C05451=1075.122,-81.429,-56.571,173.054,21.010,153.734
C05452=1075.129,-81.150,-56.583,173.055,21.011,153.734
C05453=1075.136,-80.901,-56.593,173.057,21.013,153.734
C05454=1075.142,-80.652,-56.604,173.058,21.015,153.734
C05455=1075.148,-80.401,-56.615,173.060,21.016,153.734
C05456=1075.154,-80.152,-56.626,173.061,21.018,153.734
C05457=1075.160,-79.903,-56.637,173.063,21.019,153.734
C05458=1075.166,-79.652,-56.647,173.064,21.020,153.734
C05459=1075.172,-79.403,-56.658,173.066,21.023,153.734
C05460=1075.178,-79.153,-56.669,173.068,21.024,153.734
C05461=1075.184,-78.903,-56.680,173.069,21.026,153.734
C05462=1075.190,-78.654,-56.690,173.071,21.028,153.734
C05463=1075.196,-78.404,-56.701,173.072,21.029,153.734
C05464=1075.203,-78.154,-56.712,173.074,21.030,153.734
C05465=1075.208,-77.904,-56.723,173.075,21.032,153.734
C05466=1075.214,-77.655,-56.734,173.077,21.034,153.734
C05467=1075.220,-77.405,-56.745,173.078,21.035,153.734
C05468=1075.226,-77.155,-56.756,173.080,21.037,153.735
C05469=1075.232,-76.906,-56.767,173.081,21.039,153.735
C05470=1075.239,-76.656,-56.778,173.083,21.040,153.735
C05471=1075.245,-76.406,-56.789,173.084,21.042,153.735
C05472=1075.250,-76.157,-56.800,173.086,21.044,153.735
C05473=1075.257,-75.907,-56.811,173.087,21.045,153.735
C05474=1075.263,-75.658,-56.822,173.088,21.047,153.735
C05475=1075.269,-75.408,-56.833,173.090,21.048,153.735
C05476=1075.275,-75.158,-56.845,173.092,21.050,153.735
C05477=1075.281,-74.909,-56.855,173.093,21.052,153.735
C05478=1075.287,-74.659,-56.867,173.094,21.053,153.735
C05479=1075.293,-74.409,-56.878,173.096,21.055,153.735
C05480=1075.298,-74.160,-56.888,173.097,21.057,153.735
C05481=1075.305,-73.909,-56.900,173.099,21.058,153.735
C05482=1075.310,-73.660,-56.911,173.100,21.060,153.736
C05483=1075.316,-73.410,-56.921,173.102,21.061,153.736
C05484=1075.323,-73.160,-56.933,173.103,21.063,153.736
C05485=1075.329,-72.911,-56.944,173.105,21.065,153.736
C05486=1075.334,-72.662,-56.955,173.106,21.067,153.736
C05487=1075.341,-72.412,-56.966,173.107,21.068,153.736
C05488=1075.346,-72.162,-56.977,173.109,21.070,153.736
C05489=1075.352,-71.913,-56.988,173.110,21.072,153.736
C05490=1075.358,-71.662,-57.000,173.113,21.074,153.736
C05491=1075.364,-71.413,-57.012,173.114,21.075,153.736
C05492=1075.370,-71.163,-57.023,173.115,21.077,153.736
C05493=1075.376,-70.914,-57.034,173.117,21.079,153.737
C05494=1075.382,-70.664,-57.045,173.118,21.081,153.737
C05495=1075.388,-70.414,-57.056,173.120,21.083,153.737
C05496=1075.394,-70.165,-57.067,173.121,21.084,153.737
C05497=1075.399,-69.915,-57.079,173.123,21.086,153.737
C05498=1075.405,-69.665,-57.090,173.124,21.088,153.737
C05499=1075.411,-69.416,-57.101,173.125,21.089,153.737
C05500=1075.417,-69.165,-57.112,173.127,21.091,153.737
C05501=1075.424,-68.917,-57.124,173.128,21.093,153.737
C05502=1075.429,-68.667,-57.135,173.130,21.095,153.737
C05503=1075.436,-68.417,-57.146,173.131,21.096,153.738
C05504=1075.441,-68.167,-57.157,173.132,21.098,153.738
C05505=1075.447,-67.917,-57.169,173.134,21.100,153.738
C05506=1075.453,-67.668,-57.180,173.135,21.102,153.738
C05507=1075.459,-67.418,-57.192,173.137,21.103,153.738
C05508=1075.465,-67.169,-57.203,173.138,21.105,153.738
C05509=1075.470,-66.919,-57.215,173.140,21.107,153.738
C05510=1075.477,-66.669,-57.226,173.142,21.109,153.738
C05511=1075.482,-66.419,-57.237,173.143,21.111,153.738
C05512=1075.489,-66.170,-57.249,173.145,21.112,153.738
C05513=1075.495,-65.893,-57.261,173.146,21.114,153.738
C05514=1075.502,-65.617,-57.274,173.148,21.116,153.739
C05515=1075.509,-65.341,-57.287,173.149,21.118,153.739
C05516=1075.515,-65.064,-57.299,173.151,21.121,153.739
C05517=1075.521,-64.814,-57.310,173.153,21.122,153.739
C05518=1075.527,-64.565,-57.322,173.154,21.124,153.739
C05519=1075.534,-64.315,-57.333,173.155,21.126,153.739
C05520=1075.539,-64.066,-57.345,173.157,21.127,153.739
C05521=1075.545,-63.815,-57.356,173.158,21.129,153.739
C05522=1075.551,-63.566,-57.367,173.160,21.131,153.739
C05523=1075.558,-63.316,-57.379,173.161,21.133,153.740
C05524=1075.563,-63.067,-57.390,173.162,21.135,153.740
C05525=1075.569,-62.817,-57.403,173.164,21.136,153.740
C05526=1075.575,-62.567,-57.414,173.165,21.138,153.740
C05527=1075.581,-62.317,-57.425,173.167,21.140,153.740
C05528=1075.587,-62.068,-57.436,173.169,21.142,153.740
C05529=1075.593,-61.818,-57.448,173.170,21.144,153.740
C05530=1075.599,-61.569,-57.460,173.172,21.146,153.740
C05531=1075.605,-61.319,-57.471,173.173,21.147,153.740
C05532=1075.612,-61.069,-57.483,173.175,21.149,153.741
C05533=1075.617,-60.819,-57.495,173.176,21.151,153.741
C05534=1075.624,-60.570,-57.506,173.177,21.153,153.741
C05535=1075.629,-60.320,-57.517,173.179,21.154,153.741
C05536=1075.636,-60.071,-57.529,173.180,21.156,153.741
C05537=1075.641,-59.821,-57.541,173.181,21.158,153.741
C05538=1075.648,-59.571,-57.553,173.183,21.160,153.741
C05539=1075.654,-59.321,-57.564,173.184,21.162,153.741
C05540=1075.660,-59.072,-57.576,173.186,21.164,153.742
C05541=1075.666,-58.822,-57.587,173.187,21.165,153.742
C05542=1075.672,-58.573,-57.599,173.189,21.168,153.742
C05543=1075.678,-58.323,-57.610,173.191,21.170,153.742
C05544=1075.683,-58.074,-57.622,173.192,21.172,153.742
C05545=1075.690,-57.823,-57.634,173.194,21.173,153.742
C05546=1075.696,-57.574,-57.646,173.195,21.175,153.742
C05547=1075.702,-57.325,-57.657,173.196,21.177,153.742
C05548=1075.708,-57.074,-57.669,173.198,21.178,153.742
C05549=1075.715,-56.825,-57.681,173.199,21.180,153.743
C05550=1075.720,-56.575,-57.692,173.201,21.182,153.743
C05551=1075.726,-56.326,-57.704,173.202,21.184,153.743
C05552=1075.732,-56.077,-57.716,173.203,21.186,153.743
C05553=1075.739,-55.826,-57.727,173.205,21.188,153.743
C05554=1075.745,-55.577,-57.739,173.206,21.190,153.743
C05555=1075.750,-55.327,-57.751,173.208,21.192,153.743
C05556=1075.757,-55.078,-57.763,173.210,21.193,153.743
C05557=1075.764,-54.828,-57.775,173.211,21.195,153.743
C05558=1075.769,-54.578,-57.786,173.213,21.197,153.744
C05559=1075.775,-54.329,-57.798,173.214,21.199,153.744
C05560=1075.782,-54.079,-57.810,173.215,21.201,153.744
C05561=1075.787,-53.829,-57.822,173.217,21.203,153.744
C05562=1075.794,-53.580,-57.833,173.218,21.205,153.744
C05563=1075.800,-53.330,-57.845,173.219,21.207,153.744
C05564=1075.806,-53.081,-57.858,173.221,21.208,153.744
C05565=1075.812,-52.831,-57.869,173.222,21.210,153.744
C05566=1075.819,-52.581,-57.881,173.225,21.212,153.745
C05567=1075.824,-52.332,-57.893,173.226,21.214,153.745
C05568=1075.830,-52.082,-57.904,173.227,21.216,153.745
C05569=1075.837,-51.832,-57.916,173.229,21.218,153.745
C05570=1075.843,-51.582,-57.929,173.230,21.220,153.745
C05571=1075.849,-51.333,-57.940,173.232,21.222,153.745
C05572=1075.854,-51.083,-57.952,173.233,21.224,153.745
C05573=1075.861,-50.833,-57.964,173.234,21.225,153.746
C05574=1075.867,-50.584,-57.976,173.236,21.227,153.746
C05575=1075.873,-50.335,-57.988,173.237,21.229,153.746
C05576=1075.879,-50.084,-58.000,173.238,21.231,153.746
C05577=1075.886,-49.810,-58.013,173.241,21.233,153.746
C05578=1075.892,-49.534,-58.026,173.242,21.236,153.746
C05579=1075.899,-49.259,-58.040,173.243,21.238,153.746
C05580=1075.905,-48.984,-58.053,173.245,21.240,153.747
C05581=1075.912,-48.699,-58.067,173.247,21.242,153.747
C05582=1075.919,-48.414,-58.080,173.248,21.245,153.747
C05583=1075.926,-48.130,-58.095,173.250,21.247,153.747
C05584=1075.932,-47.846,-58.108,173.251,21.249,153.747
C05585=1075.938,-47.596,-58.120,173.253,21.251,153.747
C05586=1075.944,-47.346,-58.133,173.254,21.253,153.748
C05587=1075.950,-47.097,-58.145,173.256,21.255,153.748
C05588=1075.956,-46.847,-58.157,173.258,21.257,153.748
C05589=1075.962,-46.597,-58.169,173.259,21.259,153.748
C05590=1075.968,-46.348,-58.181,173.260,21.261,153.748
C05591=1075.974,-46.098,-58.193,173.262,21.263,153.748
C05592=1075.980,-45.848,-58.206,173.263,21.265,153.748
C05593=1075.986,-45.599,-58.217,173.264,21.267,153.749
C05594=1075.992,-45.349,-58.230,173.266,21.269,153.749
C05595=1075.998,-45.099,-58.242,173.267,21.271,153.749
C05596=1076.004,-44.850,-58.254,173.269,21.273,153.749
C05597=1076.010,-44.601,-58.266,173.271,21.275,153.749
C05598=1076.015,-44.351,-58.279,173.272,21.277,153.749
C05599=1076.022,-44.101,-58.291,173.273,21.279,153.750
C05600=1076.028,-43.851,-58.304,173.275,21.281,153.750
C05601=1076.033,-43.602,-58.316,173.276,21.283,153.750
C05602=1076.040,-43.352,-58.328,173.277,21.285,153.750
C05603=1076.046,-43.103,-58.340,173.279,21.287,153.750
C05604=1076.052,-42.853,-58.353,173.280,21.289,153.750
C05605=1076.058,-42.604,-58.364,173.282,21.291,153.750
C05606=1076.064,-42.354,-58.377,173.284,21.293,153.751
C05607=1076.070,-42.104,-58.389,173.285,21.295,153.751
C05608=1076.076,-41.854,-58.401,173.286,21.297,153.751
C05609=1076.082,-41.605,-58.414,173.288,21.299,153.751
C05610=1076.087,-41.355,-58.426,173.289,21.302,153.751
C05611=1076.094,-41.106,-58.438,173.290,21.304,153.752
C05612=1076.100,-40.856,-58.451,173.291,21.306,153.752
C05613=1076.106,-40.606,-58.463,173.293,21.308,153.752
C05614=1076.112,-40.356,-58.476,173.295,21.310,153.752
C05615=1076.118,-40.107,-58.487,173.296,21.312,153.752
C05616=1076.124,-39.857,-58.500,173.298,21.314,153.752
C05617=1076.130,-39.608,-58.513,173.299,21.316,153.752
C05618=1076.136,-39.358,-58.525,173.300,21.318,153.753
C05619=1076.142,-39.108,-58.537,173.302,21.320,153.753
C05620=1076.148,-38.858,-58.550,173.303,21.322,153.753
C05621=1076.154,-38.610,-58.562,173.304,21.324,153.753
C05622=1076.160,-38.360,-58.575,173.307,21.326,153.753
C05623=1076.166,-38.110,-58.587,173.308,21.329,153.754
C05624=1076.172,-37.860,-58.600,173.309,21.330,153.754
C05625=1076.178,-37.610,-58.612,173.310,21.332,153.754
C05626=1076.183,-37.361,-58.624,173.312,21.334,153.754
C05627=1076.189,-37.111,-58.637,173.313,21.336,153.754
C05628=1076.196,-36.862,-58.650,173.315,21.338,153.754
C05629=1076.202,-36.612,-58.663,173.316,21.341,153.755
C05630=1076.207,-36.362,-58.675,173.318,21.343,153.755
C05631=1076.213,-36.113,-58.687,173.319,21.345,153.755
C05632=1076.219,-35.863,-58.700,173.321,21.347,153.755
C05633=1076.225,-35.613,-58.713,173.322,21.349,153.755
C05634=1076.231,-35.364,-58.726,173.323,21.352,153.755
C05635=1076.237,-35.115,-58.738,173.324,21.353,153.756
C05636=1076.243,-34.865,-58.750,173.326,21.355,153.756
C05637=1076.248,-34.620,-58.763,173.327,21.357,153.756
C05638=1076.254,-34.375,-58.775,173.328,21.359,153.756
C05639=1076.260,-34.131,-58.787,173.330,21.362,153.756
C05640=1076.265,-33.886,-58.800,173.332,21.364,153.757
C05641=1076.272,-33.641,-58.813,173.333,21.366,153.757
C05642=1076.278,-33.397,-58.825,173.335,21.368,153.757
C05643=1076.283,-33.152,-58.837,173.336,21.370,153.757
C05644=1076.289,-32.907,-58.850,173.337,21.372,153.757
C05645=1076.295,-32.658,-58.862,173.338,21.375,153.757
C05646=1076.301,-32.408,-58.875,173.340,21.376,153.758
C05647=1076.307,-32.158,-58.888,173.341,21.378,153.758
C05648=1076.313,-31.909,-58.900,173.342,21.380,153.758
C05649=1076.319,-31.659,-58.913,173.345,21.383,153.758
C05650=1076.325,-31.409,-58.926,173.346,21.385,153.758
C05651=1076.331,-31.159,-58.939,173.347,21.387,153.759
C05652=1076.337,-30.910,-58.951,173.348,21.389,153.759
C05653=1076.343,-30.661,-58.964,173.350,21.391,153.759
C05654=1076.349,-30.411,-58.977,173.351,21.394,153.759
C05655=1076.355,-30.162,-58.990,173.352,21.396,153.759
C05656=1076.361,-29.912,-59.003,173.355,21.398,153.759
C05657=1076.367,-29.662,-59.015,173.356,21.400,153.760
C05658=1076.373,-29.413,-59.028,173.357,21.402,153.760
C05659=1076.379,-29.163,-59.041,173.358,21.404,153.760
C05660=1076.385,-28.913,-59.054,173.360,21.406,153.760
C05661=1076.391,-28.664,-59.067,173.361,21.408,153.760
C05662=1076.397,-28.414,-59.079,173.362,21.411,153.761
C05663=1076.403,-28.165,-59.093,173.364,21.413,153.761
C05664=1076.409,-27.915,-59.105,173.366,21.415,153.761
C05665=1076.415,-27.666,-59.119,173.367,21.417,153.761
C05666=1076.421,-27.416,-59.131,173.368,21.420,153.761
C05667=1076.427,-27.166,-59.144,173.370,21.421,153.762
C05668=1076.433,-26.917,-59.157,173.371,21.423,153.762
C05669=1076.439,-26.667,-59.169,173.372,21.425,153.762
C05670=1076.445,-26.417,-59.183,173.374,21.428,153.762
C05671=1076.451,-26.167,-59.195,173.376,21.430,153.762
C05672=1076.456,-25.919,-59.209,173.377,21.433,153.763
C05673=1076.462,-25.669,-59.221,173.378,21.435,153.763
C05674=1076.468,-25.419,-59.235,173.380,21.437,153.763
C05675=1076.474,-25.170,-59.247,173.381,21.439,153.763
C05676=1076.480,-24.920,-59.260,173.382,21.441,153.763
C05677=1076.486,-24.670,-59.274,173.384,21.443,153.763
C05678=1076.492,-24.421,-59.287,173.385,21.446,153.764
C05679=1076.498,-24.171,-59.299,173.387,21.448,153.764
C05680=1076.504,-23.922,-59.313,173.388,21.450,153.764
C05681=1076.509,-23.672,-59.327,173.389,21.452,153.764
C05682=1076.515,-23.422,-59.339,173.391,21.454,153.764
C05683=1076.521,-23.173,-59.352,173.392,21.457,153.765
C05684=1076.527,-22.923,-59.365,173.394,21.459,153.765
C05685=1076.534,-22.674,-59.378,173.395,21.461,153.765
C05686=1076.539,-22.424,-59.391,173.397,21.464,153.765
C05687=1076.545,-22.174,-59.405,173.398,21.466,153.766
C05688=1076.551,-21.925,-59.418,173.399,21.468,153.766
C05689=1076.557,-21.675,-59.430,173.400,21.470,153.766
C05690=1076.563,-21.426,-59.444,173.402,21.472,153.766
C05691=1076.569,-21.176,-59.457,173.404,21.475,153.766
C05692=1076.575,-20.927,-59.470,173.405,21.477,153.767
C05693=1076.581,-20.677,-59.483,173.407,21.479,153.767
C05694=1076.586,-20.427,-59.497,173.408,21.481,153.767
C05695=1076.592,-20.178,-59.510,173.409,21.483,153.767
C05696=1076.599,-19.929,-59.523,173.410,21.486,153.767
C05697=1076.604,-19.679,-59.536,173.412,21.488,153.768
C05698=1076.610,-19.429,-59.549,173.414,21.490,153.768
C05699=1076.616,-19.180,-59.563,173.415,21.493,153.768
C05700=1076.622,-18.930,-59.575,173.416,21.494,153.768
C05701=1076.628,-18.680,-59.590,173.417,21.497,153.768
C05702=1076.634,-18.430,-59.603,173.419,21.499,153.769
C05703=1076.641,-18.181,-59.616,173.420,21.501,153.769
C05704=1076.646,-17.931,-59.629,173.422,21.504,153.769
C05705=1076.653,-17.656,-59.643,173.424,21.506,153.769
C05706=1076.659,-17.380,-59.658,173.425,21.508,153.770
C05707=1076.666,-17.105,-59.673,173.427,21.511,153.770
C05708=1076.673,-16.829,-59.688,173.428,21.513,153.770
C05709=1076.679,-16.579,-59.701,173.429,21.516,153.770
C05710=1076.684,-16.330,-59.714,173.431,21.517,153.770
C05711=1076.690,-16.080,-59.728,173.433,21.520,153.771
C05712=1076.696,-15.831,-59.741,173.434,21.522,153.771
C05713=1076.702,-15.581,-59.755,173.435,21.524,153.771
C05714=1076.708,-15.331,-59.768,173.436,21.527,153.771
C05715=1076.715,-15.082,-59.781,173.438,21.529,153.771
C05716=1076.720,-14.832,-59.795,173.439,21.531,153.772
C05717=1076.726,-14.583,-59.808,173.441,21.534,153.772
C05718=1076.732,-14.333,-59.822,173.442,21.536,153.772
C05719=1076.738,-14.083,-59.835,173.444,21.538,153.772
C05720=1076.743,-13.834,-59.849,173.445,21.541,153.773
C05721=1076.749,-13.584,-59.862,173.446,21.542,153.773
C05722=1076.755,-13.335,-59.876,173.447,21.545,153.773
C05723=1076.761,-13.086,-59.889,173.449,21.547,153.773
C05724=1076.767,-12.836,-59.903,173.451,21.550,153.773
C05725=1076.773,-12.586,-59.916,173.452,21.552,153.774
C05726=1076.779,-12.336,-59.930,173.453,21.554,153.774
C05727=1076.785,-12.087,-59.943,173.455,21.556,153.774
C05728=1076.790,-11.837,-59.957,173.456,21.559,153.774
C05729=1076.797,-11.588,-59.970,173.457,21.561,153.775
C05730=1076.802,-11.338,-59.984,173.459,21.564,153.775
C05731=1076.808,-11.089,-59.997,173.460,21.566,153.775
C05732=1076.814,-10.839,-60.011,173.462,21.568,153.775
C05733=1076.820,-10.589,-60.025,173.463,21.570,153.776
C05734=1076.826,-10.340,-60.038,173.464,21.572,153.776
C05735=1076.832,-10.091,-60.052,173.465,21.575,153.776
C05736=1076.838,-9.841,-60.066,173.468,21.577,153.776
C05737=1076.844,-9.592,-60.079,173.469,21.580,153.776
C05738=1076.849,-9.342,-60.093,173.470,21.582,153.777
C05739=1076.856,-9.093,-60.106,173.471,21.584,153.777
C05740=1076.862,-8.843,-60.120,173.473,21.586,153.777
C05741=1076.867,-8.593,-60.134,173.474,21.589,153.777
C05742=1076.873,-8.344,-60.147,173.476,21.591,153.777
C05743=1076.879,-8.094,-60.161,173.477,21.593,153.778
C05744=1076.885,-7.845,-60.174,173.479,21.595,153.778
C05745=1076.891,-7.595,-60.189,173.480,21.598,153.778
C05746=1076.897,-7.345,-60.202,173.481,21.600,153.778
C05747=1076.903,-7.096,-60.216,173.483,21.603,153.779
C05748=1076.909,-6.847,-60.229,173.485,21.605,153.779
C05749=1076.914,-6.597,-60.243,173.486,21.607,153.779
C05750=1076.921,-6.347,-60.257,173.487,21.609,153.779
C05751=1076.927,-6.097,-60.270,173.488,21.612,153.779
C05752=1076.932,-5.848,-60.284,173.489,21.614,153.780
C05753=1076.938,-5.599,-60.298,173.492,21.616,153.780
C05754=1076.945,-5.348,-60.312,173.493,21.619,153.780
C05755=1076.950,-5.099,-60.326,173.494,21.621,153.780
C05756=1076.957,-4.850,-60.340,173.495,21.623,153.781
C05757=1076.962,-4.601,-60.354,173.497,21.625,153.781
C05758=1076.969,-4.351,-60.367,173.498,21.628,153.781
C05759=1076.974,-4.101,-60.381,173.500,21.630,153.781
C05760=1076.980,-3.851,-60.395,173.501,21.633,153.782
C05761=1076.986,-3.602,-60.408,173.503,21.634,153.782
C05762=1076.992,-3.353,-60.423,173.504,21.637,153.782
C05763=1076.998,-3.103,-60.437,173.505,21.639,153.782
C05764=1077.004,-2.854,-60.450,173.506,21.641,153.782
C05765=1077.010,-2.604,-60.464,173.508,21.644,153.783
C05766=1077.016,-2.354,-60.478,173.510,21.646,153.783
C05767=1077.021,-2.104,-60.492,173.511,21.649,153.783
C05768=1077.027,-1.855,-60.507,173.512,21.651,153.783
C05769=1077.033,-1.578,-60.522,173.514,21.654,153.784
C05770=1077.040,-1.300,-60.538,173.515,21.657,153.784
C05771=1077.046,-1.023,-60.553,173.516,21.659,153.784
C05772=1077.053,-0.746,-60.569,173.518,21.662,153.785
C05773=1077.058,-0.496,-60.583,173.520,21.664,153.785
C05774=1077.064,-0.247,-60.597,173.521,21.666,153.785
C05775=1077.070,0.002,-60.610,173.522,21.669,153.785
C05776=1077.076,0.252,-60.625,173.524,21.671,153.785
C05777=1077.082,0.501,-60.639,173.526,21.674,153.786
C05778=1077.088,0.751,-60.653,173.527,21.676,153.786
C05779=1077.093,1.000,-60.667,173.528,21.678,153.786
C05780=1077.099,1.251,-60.681,173.529,21.681,153.786
C05781=1077.105,1.500,-60.696,173.531,21.683,153.787
C05782=1077.110,1.749,-60.710,173.533,21.685,153.787
C05783=1077.117,1.999,-60.723,173.534,21.688,153.787
C05784=1077.123,2.248,-60.738,173.535,21.690,153.787
C05785=1077.128,2.498,-60.752,173.536,21.692,153.788
C05786=1077.134,2.747,-60.766,173.537,21.695,153.788
C05787=1077.140,2.997,-60.781,173.540,21.698,153.788
C05788=1077.146,3.247,-60.794,173.541,21.700,153.788
C05789=1077.151,3.496,-60.808,173.542,21.702,153.789
C05790=1077.158,3.746,-60.823,173.543,21.705,153.789
C05791=1077.163,3.995,-60.837,173.545,21.707,153.789
C05792=1077.170,4.244,-60.851,173.547,21.709,153.789
C05793=1077.176,4.494,-60.865,173.548,21.711,153.789
C05794=1077.181,4.744,-60.879,173.549,21.714,153.790
C05795=1077.187,4.993,-60.894,173.550,21.716,153.790
C05796=1077.193,5.243,-60.908,173.552,21.718,153.790
C05797=1077.199,5.492,-60.923,173.554,21.721,153.790
C05798=1077.204,5.742,-60.936,173.555,21.724,153.791
C05799=1077.211,5.991,-60.951,173.556,21.726,153.791
C05800=1077.216,6.241,-60.965,173.557,21.728,153.791
C05801=1077.222,6.490,-60.979,173.559,21.730,153.792
C05802=1077.228,6.740,-60.994,173.560,21.732,153.792
C05803=1077.234,6.990,-61.008,173.562,21.735,153.792
C05804=1077.239,7.239,-61.022,173.563,21.738,153.792
C05805=1077.245,7.489,-61.037,173.565,21.740,153.792
C05806=1077.252,7.738,-61.051,173.566,21.742,153.793
C05807=1077.258,7.988,-61.065,173.567,21.745,153.793
C05808=1077.264,8.237,-61.079,173.569,21.747,153.793
C05809=1077.269,8.486,-61.093,173.570,21.750,153.793
C05810=1077.276,8.736,-61.108,173.572,21.752,153.794
C05811=1077.281,8.985,-61.123,173.573,21.754,153.794
C05812=1077.288,9.235,-61.137,173.574,21.756,153.794
C05813=1077.293,9.484,-61.152,173.576,21.759,153.794
C05814=1077.299,9.735,-61.166,173.577,21.761,153.795
C05815=1077.305,9.983,-61.181,173.579,21.764,153.795
C05816=1077.311,10.233,-61.194,173.580,21.766,153.795
C05817=1077.317,10.483,-61.209,173.581,21.768,153.795
C05818=1077.323,10.732,-61.224,173.583,21.771,153.796
C05819=1077.329,10.982,-61.238,173.585,21.773,153.796
C05820=1077.335,11.231,-61.253,173.586,21.775,153.796
C05821=1077.341,11.481,-61.267,173.587,21.778,153.796
C05822=1077.347,11.730,-61.282,173.588,21.780,153.797
C05823=1077.353,11.980,-61.296,173.590,21.783,153.797
C05824=1077.358,12.229,-61.310,173.592,21.785,153.797
C05825=1077.365,12.479,-61.325,173.593,21.787,153.797
C05826=1077.371,12.728,-61.340,173.594,21.790,153.798
C05827=1077.376,12.978,-61.354,173.595,21.792,153.798
C05828=1077.382,13.227,-61.369,173.598,21.794,153.798
C05829=1077.388,13.476,-61.383,173.599,21.797,153.798
C05830=1077.394,13.726,-61.397,173.600,21.799,153.799
C05831=1077.400,13.975,-61.412,173.601,21.801,153.799
C05832=1077.406,14.225,-61.427,173.602,21.804,153.799
C05833=1077.413,14.505,-61.443,173.604,21.807,153.799
C05834=1077.419,14.783,-61.460,173.606,21.809,153.800
C05835=1077.426,15.063,-61.476,173.608,21.812,153.800
C05836=1077.432,15.342,-61.493,173.609,21.814,153.800
C05837=1077.438,15.592,-61.507,173.610,21.817,153.800
C05838=1077.444,15.842,-61.522,173.612,21.819,153.801
C05839=1077.450,16.091,-61.536,173.614,21.822,153.801
C05840=1077.456,16.340,-61.551,173.615,21.824,153.801
C05841=1077.461,16.590,-61.566,173.616,21.827,153.801
C05842=1077.467,16.840,-61.581,173.617,21.829,153.802
C05843=1077.473,17.089,-61.595,173.619,21.832,153.802
C05844=1077.480,17.338,-61.610,173.620,21.834,153.802
C05845=1077.485,17.587,-61.625,173.622,21.836,153.802
C05846=1077.491,17.838,-61.640,173.623,21.838,153.803
C05847=1077.496,18.087,-61.654,173.625,21.841,153.803
C05848=1077.503,18.337,-61.669,173.626,21.844,153.803
C05849=1077.509,18.586,-61.684,173.628,21.846,153.803
C05850=1077.514,18.836,-61.699,173.629,21.848,153.804
C05851=1077.520,19.084,-61.714,173.630,21.851,153.804
C05852=1077.526,19.335,-61.728,173.632,21.853,153.804
C05853=1077.532,19.584,-61.743,173.633,21.855,153.804
C05854=1077.538,19.834,-61.758,173.635,21.858,153.805
C05855=1077.543,20.083,-61.773,173.636,21.860,153.805
C05856=1077.550,20.332,-61.788,173.637,21.862,153.805
C05857=1077.555,20.581,-61.802,173.639,21.865,153.805
C05858=1077.561,20.831,-61.818,173.640,21.868,153.806
C05859=1077.567,21.080,-61.832,173.642,21.870,153.806
C05860=1077.573,21.330,-61.848,173.643,21.872,153.806
C05861=1077.578,21.579,-61.863,173.644,21.874,153.806
C05862=1077.584,21.829,-61.877,173.646,21.877,153.807
C05863=1077.590,22.079,-61.892,173.647,21.880,153.807
C05864=1077.596,22.328,-61.907,173.649,21.882,153.807
C05865=1077.602,22.578,-61.922,173.650,21.884,153.807
C05866=1077.607,22.827,-61.937,173.652,21.887,153.808
C05867=1077.614,23.077,-61.952,173.653,21.890,153.808
C05868=1077.619,23.326,-61.967,173.655,21.892,153.808
C05869=1077.625,23.576,-61.982,173.656,21.894,153.808
C05870=1077.631,23.825,-61.997,173.657,21.896,153.809
C05871=1077.637,24.075,-62.012,173.659,21.899,153.809
C05872=1077.643,24.324,-62.027,173.660,21.901,153.809
C05873=1077.649,24.573,-62.042,173.662,21.904,153.809
C05874=1077.654,24.823,-62.057,173.663,21.906,153.810
C05875=1077.660,25.072,-62.072,173.665,21.909,153.810
C05876=1077.666,25.322,-62.087,173.666,21.911,153.810
C05877=1077.672,25.572,-62.102,173.667,21.913,153.810
C05878=1077.678,25.821,-62.117,173.669,21.916,153.811
C05879=1077.684,26.070,-62.133,173.670,21.918,153.811
C05880=1077.690,26.320,-62.148,173.672,21.921,153.811
C05881=1077.695,26.569,-62.163,173.673,21.923,153.811
C05882=1077.702,26.819,-62.178,173.674,21.926,153.812
C05883=1077.707,27.068,-62.193,173.676,21.928,153.812
C05884=1077.713,27.318,-62.208,173.678,21.930,153.812
C05885=1077.719,27.567,-62.223,173.679,21.933,153.812
C05886=1077.725,27.817,-62.239,173.680,21.935,153.813
C05887=1077.731,28.066,-62.253,173.682,21.937,153.813
C05888=1077.737,28.316,-62.269,173.683,21.940,153.813
C05889=1077.743,28.565,-62.284,173.685,21.943,153.813
C05890=1077.748,28.815,-62.300,173.686,21.945,153.814
C05891=1077.755,29.064,-62.315,173.687,21.947,153.814
C05892=1077.760,29.313,-62.330,173.689,21.949,153.814
C05893=1077.765,29.563,-62.346,173.691,21.952,153.814
C05894=1077.771,29.812,-62.360,173.692,21.955,153.815
C05895=1077.777,30.062,-62.376,173.693,21.957,153.815
C05896=1077.783,30.311,-62.391,173.694,21.959,153.815
C05897=1077.790,30.592,-62.408,173.696,21.963,153.816
C05898=1077.796,30.873,-62.425,173.697,21.965,153.816
C05899=1077.803,31.153,-62.443,173.699,21.968,153.816
C05900=1077.809,31.434,-62.461,173.701,21.970,153.816
C05901=1077.815,31.683,-62.475,173.703,21.973,153.817
C05902=1077.820,31.933,-62.491,173.704,21.976,153.817
C05903=1077.827,32.182,-62.507,173.705,21.978,153.817
C05904=1077.832,32.432,-62.522,173.706,21.980,153.817
C05905=1077.838,32.681,-62.537,173.709,21.983,153.818
C05906=1077.844,32.931,-62.552,173.710,21.986,153.818
C05907=1077.850,33.180,-62.568,173.711,21.987,153.818
C05908=1077.856,33.429,-62.583,173.712,21.990,153.818
C05909=1077.862,33.679,-62.599,173.714,21.993,153.819
C05910=1077.867,33.928,-62.615,173.716,21.995,153.819
C05911=1077.873,34.178,-62.629,173.717,21.997,153.819
C05912=1077.879,34.428,-62.645,173.718,22.000,153.820
C05913=1077.885,34.677,-62.661,173.719,22.002,153.820
C05914=1077.891,34.926,-62.676,173.721,22.005,153.820
C05915=1077.896,35.176,-62.691,173.723,22.007,153.820
C05916=1077.902,35.425,-62.708,173.724,22.009,153.821
C05917=1077.909,35.675,-62.723,173.725,22.012,153.821
C05918=1077.914,35.924,-62.738,173.727,22.015,153.821
C05919=1077.920,36.174,-62.754,173.729,22.017,153.821
C05920=1077.926,36.423,-62.769,173.730,22.019,153.822
C05921=1077.932,36.673,-62.785,173.731,22.021,153.822
C05922=1077.937,36.922,-62.800,173.733,22.024,153.822
C05923=1077.943,37.172,-62.815,173.734,22.026,153.822
C05924=1077.949,37.421,-62.832,173.736,22.029,153.823
C05925=1077.955,37.671,-62.847,173.737,22.031,153.823
C05926=1077.961,37.919,-62.862,173.739,22.034,153.823
C05927=1077.967,38.169,-62.878,173.740,22.036,153.823
C05928=1077.973,38.418,-62.894,173.741,22.038,153.824
C05929=1077.978,38.668,-62.910,173.743,22.041,153.824
C05930=1077.984,38.917,-62.926,173.745,22.044,153.824
C05931=1077.989,39.167,-62.941,173.746,22.046,153.824
C05932=1077.996,39.416,-62.957,173.747,22.048,153.825
C05933=1078.002,39.666,-62.972,173.749,22.051,153.825
C05934=1078.007,39.915,-62.988,173.751,22.053,153.825
C05935=1078.013,40.165,-63.004,173.752,22.056,153.825
C05936=1078.019,40.414,-63.020,173.753,22.058,153.826
C05937=1078.024,40.664,-63.036,173.754,22.060,153.826
C05938=1078.030,40.912,-63.051,173.756,22.063,153.826
C05939=1078.036,41.162,-63.066,173.758,22.066,153.826
C05940=1078.042,41.412,-63.083,173.759,22.068,153.827
C05941=1078.048,41.662,-63.098,173.760,22.071,153.827
C05942=1078.054,41.911,-63.115,173.762,22.073,153.827
C05943=1078.059,42.160,-63.130,173.763,22.075,153.827
C05944=1078.065,42.410,-63.146,173.765,22.078,153.828
C05945=1078.071,42.659,-63.162,173.766,22.080,153.828
C05946=1078.077,42.909,-63.177,173.768,22.083,153.828
C05947=1078.083,43.158,-63.193,173.769,22.085,153.828
C05948=1078.088,43.407,-63.209,173.771,22.087,153.829
C05949=1078.094,43.657,-63.225,173.773,22.090,153.829
C05950=1078.100,43.906,-63.241,173.774,22.092,153.829
C05951=1078.105,44.156,-63.257,173.775,22.095,153.830
C05952=1078.111,44.405,-63.273,173.776,22.097,153.830
C05953=1078.117,44.654,-63.289,173.778,22.100,153.830
C05954=1078.122,44.904,-63.304,173.780,22.102,153.830
C05955=1078.128,45.153,-63.321,173.781,22.105,153.831
C05956=1078.134,45.403,-63.337,173.782,22.107,153.831
C05957=1078.140,45.652,-63.352,173.784,22.110,153.831
C05958=1078.145,45.901,-63.369,173.786,22.112,153.831
C05959=1078.150,46.151,-63.385,173.787,22.115,153.832
C05960=1078.156,46.401,-63.401,173.788,22.117,153.832
C05961=1078.163,46.681,-63.418,173.790,22.120,153.832
C05962=1078.169,46.961,-63.437,173.792,22.123,153.832
C05963=1078.176,47.243,-63.456,173.793,22.126,153.833
C05964=1078.182,47.523,-63.473,173.795,22.129,153.833
C05965=1078.188,47.773,-63.489,173.796,22.131,153.833
C05966=1078.194,48.022,-63.505,173.798,22.133,153.834
C05967=1078.199,48.271,-63.522,173.799,22.135,153.834
C05968=1078.205,48.520,-63.538,173.801,22.138,153.834
C05969=1078.210,48.770,-63.553,173.802,22.141,153.834
C05970=1078.216,49.020,-63.570,173.803,22.143,153.835
C05971=1078.222,49.269,-63.586,173.806,22.146,153.835
C05972=1078.228,49.518,-63.602,173.807,22.148,153.835
C05973=1078.234,49.768,-63.618,173.808,22.150,153.836
C05974=1078.239,50.016,-63.634,173.809,22.153,153.836
C05975=1078.244,50.267,-63.650,173.811,22.156,153.836
C05976=1078.250,50.516,-63.667,173.813,22.158,153.836
C05977=1078.256,50.765,-63.683,173.814,22.160,153.837
C05978=1078.262,51.015,-63.699,173.816,22.163,153.837
C05979=1078.268,51.264,-63.715,173.817,22.165,153.837
C05980=1078.274,51.513,-63.732,173.818,22.168,153.837
C05981=1078.280,51.763,-63.748,173.820,22.170,153.838
C05982=1078.285,52.013,-63.764,173.822,22.173,153.838
C05983=1078.291,52.262,-63.780,173.823,22.175,153.838
C05984=1078.296,52.511,-63.796,173.824,22.178,153.838
C05985=1078.302,52.760,-63.812,173.826,22.179,153.839
C05986=1078.308,53.010,-63.829,173.828,22.182,153.839
C05987=1078.314,53.259,-63.845,173.829,22.185,153.839
C05988=1078.320,53.508,-63.861,173.830,22.187,153.839
C05989=1078.325,53.758,-63.878,173.833,22.190,153.840
C05990=1078.331,54.007,-63.894,173.834,22.192,153.840
C05991=1078.337,54.257,-63.911,173.835,22.194,153.840
C05992=1078.343,54.506,-63.927,173.836,22.197,153.840
C05993=1078.349,54.756,-63.943,173.838,22.199,153.841
C05994=1078.354,55.005,-63.960,173.840,22.202,153.841
C05995=1078.360,55.255,-63.976,173.841,22.204,153.841
C05996=1078.366,55.504,-63.993,173.843,22.207,153.841
C05997=1078.372,55.753,-64.009,173.844,22.209,153.842
C05998=1078.378,56.003,-64.025,173.846,22.211,153.842
C05999=1078.383,56.252,-64.042,173.848,22.214,153.842
C06000=1078.389,56.502,-64.058,173.849,22.217,153.842
C06001=1078.395,56.751,-64.074,173.850,22.219,153.843
C06002=1078.401,57.000,-64.091,173.851,22.221,153.843
C06003=1078.407,57.250,-64.107,173.853,22.224,153.843
C06004=1078.412,57.499,-64.124,173.855,22.226,153.843
C06005=1078.418,57.749,-64.140,173.856,22.228,153.844
C06006=1078.424,57.998,-64.156,173.858,22.231,153.844
C06007=1078.430,58.247,-64.173,173.860,22.233,153.844
C06008=1078.435,58.497,-64.189,173.861,22.235,153.844
C06009=1078.442,58.746,-64.206,173.862,22.238,153.845
C06010=1078.448,58.995,-64.223,173.864,22.241,153.845
C06011=1078.454,59.244,-64.239,173.865,22.243,153.845
C06012=1078.459,59.494,-64.256,173.867,22.245,153.845
C06013=1078.465,59.743,-64.272,173.869,22.248,153.846
C06014=1078.471,59.993,-64.289,173.870,22.250,153.846
C06015=1078.477,60.243,-64.305,173.871,22.252,153.846
C06016=1078.483,60.492,-64.322,173.873,22.255,153.846
C06017=1078.489,60.741,-64.339,173.875,22.257,153.847
C06018=1078.495,60.991,-64.355,173.876,22.259,153.847
C06019=1078.501,61.240,-64.371,173.877,22.262,153.847
C06020=1078.506,61.490,-64.388,173.880,22.264,153.847
C06021=1078.512,61.738,-64.405,173.881,22.267,153.848
C06022=1078.518,61.988,-64.421,173.882,22.269,153.848
C06023=1078.524,62.237,-64.438,173.884,22.271,153.848
C06024=1078.530,62.487,-64.455,173.885,22.274,153.848
C06025=1078.537,62.767,-64.473,173.888,22.277,153.849
C06026=1078.543,63.047,-64.492,173.889,22.279,153.849
C06027=1078.550,63.328,-64.511,173.891,22.282,153.849
C06028=1078.556,63.608,-64.529,173.892,22.284,153.849
C06029=1078.562,63.858,-64.546,173.894,22.287,153.849
C06030=1078.569,64.107,-64.563,173.896,22.289,153.850
C06031=1078.574,64.357,-64.580,173.897,22.292,153.850
C06032=1078.580,64.606,-64.596,173.899,22.294,153.850
C06033=1078.585,64.855,-64.614,173.900,22.296,153.851
C06034=1078.591,65.105,-64.630,173.901,22.299,153.851
C06035=1078.597,65.354,-64.647,173.904,22.301,153.851
C06036=1078.603,65.603,-64.664,173.905,22.304,153.851
C06037=1078.608,65.853,-64.681,173.906,22.306,153.852
C06038=1078.614,66.102,-64.697,173.908,22.308,153.852
C06039=1078.620,66.352,-64.715,173.910,22.311,153.852
C06040=1078.626,66.601,-64.731,173.911,22.313,153.852
C06041=1078.631,66.851,-64.748,173.912,22.316,153.853
C06042=1078.638,67.099,-64.765,173.914,22.318,153.853
C06043=1078.643,67.349,-64.782,173.916,22.320,153.853
C06044=1078.649,67.598,-64.799,173.917,22.323,153.853
C06045=1078.654,67.848,-64.816,173.919,22.325,153.853
C06046=1078.661,68.098,-64.832,173.920,22.328,153.854
C06047=1078.666,68.347,-64.850,173.922,22.330,153.854
C06048=1078.672,68.596,-64.866,173.924,22.332,153.854
C06049=1078.678,68.845,-64.884,173.925,22.335,153.854
C06050=1078.684,69.094,-64.900,173.926,22.337,153.855
C06051=1078.689,69.343,-64.917,173.929,22.340,153.855
C06052=1078.694,69.593,-64.934,173.930,22.342,153.855
C06053=1078.701,69.843,-64.952,173.931,22.344,153.855
C06054=1078.707,70.092,-64.968,173.933,22.347,153.856
C06055=1078.713,70.341,-64.985,173.934,22.349,153.856
C06056=1078.718,70.591,-65.002,173.936,22.352,153.856
C06057=1078.724,70.840,-65.020,173.938,22.354,153.856
C06058=1078.729,71.089,-65.036,173.939,22.356,153.857
C06059=1078.736,71.339,-65.054,173.940,22.359,153.857
C06060=1078.741,71.588,-65.071,173.943,22.362,153.857
C06061=1078.747,71.837,-65.088,173.944,22.364,153.857
C06062=1078.752,72.087,-65.105,173.945,22.366,153.858
C06063=1078.758,72.336,-65.122,173.947,22.369,153.858
C06064=1078.764,72.586,-65.139,173.949,22.371,153.858
C06065=1078.770,72.835,-65.156,173.950,22.373,153.858
C06066=1078.775,73.084,-65.174,173.952,22.376,153.859
C06067=1078.781,73.334,-65.191,173.953,22.378,153.859
C06068=1078.787,73.582,-65.208,173.955,22.380,153.859
C06069=1078.793,73.833,-65.225,173.957,22.383,153.859
C06070=1078.798,74.082,-65.243,173.958,22.385,153.860
C06071=1078.804,74.330,-65.260,173.959,22.388,153.860
C06072=1078.810,74.580,-65.276,173.961,22.390,153.860
C06073=1078.815,74.829,-65.294,173.963,22.392,153.860
C06074=1078.821,75.079,-65.312,173.964,22.395,153.861
C06075=1078.827,75.328,-65.328,173.966,22.398,153.861
C06076=1078.833,75.577,-65.346,173.968,22.399,153.861
C06077=1078.838,75.826,-65.363,173.969,22.402,153.861
C06078=1078.844,76.077,-65.381,173.971,22.405,153.862
C06079=1078.850,76.325,-65.397,173.972,22.407,153.862
C06080=1078.856,76.574,-65.415,173.973,22.409,153.862
C06081=1078.861,76.824,-65.432,173.976,22.412,153.862
C06082=1078.867,77.074,-65.450,173.977,22.414,153.862
C06083=1078.873,77.323,-65.467,173.978,22.416,153.863
C06084=1078.879,77.572,-65.484,173.981,22.419,153.863
C06085=1078.885,77.822,-65.502,173.982,22.421,153.863
C06086=1078.890,78.071,-65.519,173.984,22.424,153.863
C06087=1078.896,78.320,-65.537,173.985,22.426,153.864
C06088=1078.901,78.570,-65.554,173.986,22.428,153.864
C06089=1078.908,78.850,-65.574,173.989,22.431,153.864
C06090=1078.915,79.130,-65.593,173.991,22.434,153.864
C06091=1078.921,79.410,-65.613,173.992,22.436,153.865
C06092=1078.928,79.691,-65.632,173.994,22.439,153.865
C06093=1078.933,79.940,-65.650,173.995,22.442,153.865
C06094=1078.939,80.189,-65.667,173.998,22.444,153.865
C06095=1078.944,80.439,-65.684,173.999,22.446,153.866
C06096=1078.950,80.688,-65.702,174.000,22.449,153.866
C06097=1078.956,80.937,-65.720,174.002,22.451,153.866
C06098=1078.961,81.187,-65.737,174.003,22.453,153.866
C06099=1078.967,81.436,-65.755,174.005,22.456,153.867
C06100=1078.973,81.685,-65.773,174.007,22.458,153.867
C06101=1078.978,81.934,-65.790,174.008,22.461,153.867
C06102=1078.984,82.184,-65.807,174.009,22.463,153.867
C06103=1078.990,82.434,-65.825,174.012,22.465,153.868
C06104=1078.995,82.683,-65.843,174.013,22.468,153.868
C06105=1079.001,82.932,-65.860,174.015,22.471,153.868
C06106=1079.007,83.182,-65.878,174.016,22.473,153.868
C06107=1079.012,83.431,-65.896,174.018,22.475,153.869
C06108=1079.018,83.680,-65.913,174.020,22.477,153.869
C06109=1079.024,83.929,-65.931,174.021,22.480,153.869
C06110=1079.030,84.178,-65.949,174.022,22.482,153.869
C06111=1079.035,84.427,-65.966,174.025,22.484,153.869
C06112=1079.041,84.677,-65.984,174.026,22.487,153.870
C06113=1079.047,84.926,-66.002,174.028,22.489,153.870
C06114=1079.053,85.176,-66.020,174.029,22.492,153.870
C06115=1079.058,85.425,-66.037,174.031,22.494,153.871
C06116=1079.064,85.674,-66.055,174.033,22.496,153.871
C06117=1079.070,85.924,-66.073,174.034,22.499,153.871
C06118=1079.076,86.173,-66.091,174.036,22.501,153.871
C06119=1079.081,86.422,-66.108,174.038,22.503,153.871
C06120=1079.087,86.672,-66.126,174.039,22.506,153.872
C06121=1079.093,86.921,-66.144,174.041,22.508,153.872
C06122=1079.099,87.170,-66.162,174.043,22.511,153.872
C06123=1079.104,87.419,-66.179,174.044,22.513,153.872
C06124=1079.110,87.668,-66.197,174.046,22.515,153.873
C06125=1079.116,87.918,-66.215,174.047,22.517,153.873
C06126=1079.122,88.167,-66.232,174.049,22.520,153.873
C06127=1079.127,88.417,-66.251,174.051,22.522,153.873
C06128=1079.133,88.666,-66.269,174.052,22.524,153.873
C06129=1079.139,88.915,-66.287,174.055,22.527,153.874
C06130=1079.144,89.165,-66.304,174.056,22.529,153.874
C06131=1079.150,89.414,-66.322,174.057,22.531,153.874
C06132=1079.156,89.663,-66.340,174.059,22.534,153.874
C06133=1079.162,89.912,-66.358,174.060,22.536,153.875
C06134=1079.168,90.162,-66.375,174.063,22.539,153.875
C06135=1079.173,90.410,-66.394,174.064,22.541,153.875
C06136=1079.180,90.660,-66.412,174.065,22.543,153.875
C06137=1079.185,90.909,-66.429,174.068,22.546,153.875
C06138=1079.191,91.159,-66.448,174.069,22.548,153.876
C06139=1079.196,91.408,-66.465,174.071,22.550,153.876
C06140=1079.202,91.657,-66.484,174.072,22.552,153.876
C06141=1079.208,91.907,-66.502,174.074,22.555,153.876
C06142=1079.213,92.156,-66.520,174.076,22.558,153.877
C06143=1079.219,92.406,-66.538,174.077,22.560,153.877
C06144=1079.224,92.655,-66.555,174.079,22.562,153.877
C06145=1079.231,92.904,-66.574,174.081,22.564,153.877
C06146=1079.236,93.153,-66.592,174.082,22.567,153.878
C06147=1079.242,93.403,-66.610,174.084,22.569,153.878
C06148=1079.248,93.651,-66.628,174.086,22.571,153.878
C06149=1079.253,93.901,-66.647,174.088,22.574,153.878
C06150=1079.258,94.150,-66.664,174.089,22.576,153.878
C06151=1079.265,94.400,-66.682,174.090,22.579,153.879
C06152=1079.270,94.649,-66.701,174.093,22.581,153.879
C06153=1079.276,94.930,-66.721,174.095,22.584,153.879
C06154=1079.283,95.210,-66.741,174.096,22.586,153.879
C06155=1079.290,95.490,-66.762,174.098,22.589,153.880
C06156=1079.296,95.771,-66.782,174.100,22.592,153.880
C06157=1079.301,96.020,-66.801,174.102,22.594,153.880
C06158=1079.307,96.269,-66.819,174.103,22.596,153.880
C06159=1079.313,96.518,-66.837,174.105,22.598,153.880
C06160=1079.318,96.768,-66.856,174.106,22.601,153.881
C06161=1079.324,97.017,-66.873,174.109,22.603,153.881
C06162=1079.330,97.266,-66.892,174.110,22.605,153.881
C06163=1079.335,97.515,-66.910,174.112,22.608,153.881
C06164=1079.341,97.764,-66.929,174.113,22.610,153.882
C06165=1079.347,98.013,-66.946,174.115,22.612,153.882
C06166=1079.353,98.263,-66.966,174.117,22.615,153.882
C06167=1079.358,98.512,-66.983,174.118,22.617,153.882
C06168=1079.364,98.762,-67.002,174.121,22.619,153.882
C06169=1079.370,99.011,-67.020,174.122,22.622,153.883
C06170=1079.376,99.260,-67.038,174.124,22.624,153.883
C06171=1079.381,99.510,-67.057,174.126,22.626,153.883
C06172=1079.387,99.759,-67.075,174.127,22.628,153.883
C06173=1079.393,100.008,-67.093,174.129,22.631,153.884
C06174=1079.398,100.257,-67.112,174.130,22.633,153.884
C06175=1079.404,100.506,-67.130,174.133,22.636,153.884
C06176=1079.410,100.756,-67.149,174.134,22.638,153.884
C06177=1079.416,101.005,-67.167,174.136,22.640,153.884
C06178=1079.422,101.254,-67.186,174.138,22.642,153.885
C06179=1079.427,101.503,-67.204,174.139,22.644,153.885
C06180=1079.433,101.752,-67.222,174.141,22.647,153.885
C06181=1079.439,102.002,-67.241,174.143,22.649,153.885
C06182=1079.444,102.251,-67.260,174.145,22.652,153.885
C06183=1079.450,102.501,-67.278,174.146,22.654,153.886
C06184=1079.455,102.750,-67.297,174.148,22.656,153.886
C06185=1079.461,102.999,-67.315,174.150,22.658,153.886
C06186=1079.466,103.248,-67.333,174.152,22.661,153.886
C06187=1079.473,103.497,-67.352,174.153,22.663,153.886
C06188=1079.478,103.747,-67.371,174.154,22.665,153.887
C06189=1079.483,103.996,-67.389,174.157,22.668,153.887
C06190=1079.489,104.245,-67.408,174.158,22.670,153.887
C06191=1079.494,104.494,-67.426,174.160,22.672,153.887
C06192=1079.501,104.743,-67.445,174.161,22.675,153.888
C06193=1079.506,104.993,-67.464,174.164,22.677,153.888
C06194=1079.511,105.242,-67.482,174.165,22.680,153.888
C06195=1079.518,105.491,-67.501,174.167,22.682,153.888
C06196=1079.523,105.741,-67.520,174.169,22.684,153.888
C06197=1079.529,105.989,-67.539,174.170,22.686,153.889
C06198=1079.534,106.239,-67.557,174.172,22.689,153.889
C06199=1079.540,106.488,-67.576,174.174,22.691,153.889
C06200=1079.546,106.737,-67.595,174.176,22.693,153.889
C06201=1079.552,106.987,-67.614,174.177,22.696,153.890
C06202=1079.556,107.236,-67.632,174.179,22.698,153.890
C06203=1079.563,107.485,-67.651,174.181,22.700,153.890
C06204=1079.569,107.735,-67.670,174.183,22.703,153.890
C06205=1079.574,107.984,-67.689,174.184,22.704,153.890
C06206=1079.580,108.233,-67.707,174.187,22.707,153.891
C06207=1079.585,108.482,-67.726,174.188,22.709,153.891
C06208=1079.592,108.732,-67.745,174.189,22.711,153.891
C06209=1079.597,108.980,-67.763,174.191,22.714,153.891
C06210=1079.603,109.230,-67.783,174.193,22.716,153.891
C06211=1079.609,109.479,-67.801,174.195,22.718,153.892
C06212=1079.614,109.728,-67.820,174.196,22.720,153.892
C06213=1079.620,109.978,-67.839,174.199,22.723,153.892
C06214=1079.626,110.227,-67.857,174.200,22.725,153.892
C06215=1079.632,110.476,-67.877,174.202,22.727,153.892
C06216=1079.637,110.725,-67.896,174.204,22.730,153.893
C06217=1079.644,111.006,-67.917,174.206,22.732,153.893
C06218=1079.650,111.286,-67.938,174.208,22.735,153.893
C06219=1079.656,111.566,-67.959,174.210,22.738,153.893
C06220=1079.662,111.847,-67.981,174.212,22.740,153.893
C06221=1079.669,112.096,-67.999,174.214,22.742,153.894
C06222=1079.674,112.345,-68.019,174.215,22.744,153.894
C06223=1079.680,112.595,-68.038,174.217,22.747,153.894
C06224=1079.685,112.843,-68.057,174.219,22.749,153.894
C06225=1079.691,113.093,-68.076,174.221,22.751,153.894
C06226=1079.697,113.342,-68.095,174.222,22.753,153.895
C06227=1079.703,113.591,-68.114,174.225,22.756,153.895
C06228=1079.708,113.840,-68.133,174.226,22.758,153.895
C06229=1079.714,114.090,-68.152,174.228,22.761,153.895
C06230=1079.719,114.339,-68.171,174.230,22.763,153.895
C06231=1079.725,114.588,-68.191,174.232,22.765,153.896
C06232=1079.730,114.837,-68.209,174.233,22.767,153.896
C06233=1079.736,115.087,-68.229,174.235,22.770,153.896
C06234=1079.742,115.336,-68.248,174.237,22.772,153.896
C06235=1079.747,115.585,-68.267,174.239,22.774,153.896
C06236=1079.752,115.834,-68.286,174.240,22.777,153.897
C06237=1079.758,116.084,-68.305,174.243,22.779,153.897
C06238=1079.764,116.333,-68.325,174.244,22.781,153.897
C06239=1079.769,116.582,-68.343,174.246,22.784,153.897
C06240=1079.775,116.831,-68.363,174.248,22.785,153.898
C06241=1079.780,117.081,-68.382,174.250,22.788,153.898
C06242=1079.786,117.330,-68.401,174.251,22.790,153.898
C06243=1079.791,117.578,-68.421,174.253,22.792,153.898
C06244=1079.797,117.828,-68.440,174.255,22.795,153.898
C06245=1079.803,118.077,-68.459,174.257,22.797,153.899
C06246=1079.808,118.326,-68.478,174.258,22.800,153.899
C06247=1079.814,118.576,-68.498,174.261,22.802,153.899
C06248=1079.819,118.825,-68.517,174.262,22.804,153.899
C06249=1079.825,119.073,-68.537,174.264,22.807,153.899
C06250=1079.831,119.323,-68.556,174.266,22.808,153.900
C06251=1079.836,119.572,-68.575,174.268,22.811,153.900
C06252=1079.842,119.822,-68.594,174.269,22.813,153.900
C06253=1079.847,120.070,-68.613,174.271,22.815,153.900
C06254=1079.853,120.319,-68.633,174.273,22.817,153.900
C06255=1079.859,120.569,-68.652,174.275,22.820,153.901
C06256=1079.865,120.818,-68.672,174.276,22.822,153.901
C06257=1079.870,121.068,-68.691,174.279,22.824,153.901
C06258=1079.876,121.316,-68.711,174.280,22.827,153.901
C06259=1079.881,121.565,-68.730,174.282,22.829,153.901
C06260=1079.886,121.815,-68.750,174.284,22.831,153.901
C06261=1079.892,122.064,-68.769,174.286,22.834,153.902
C06262=1079.898,122.313,-68.789,174.288,22.836,153.902
C06263=1079.904,122.563,-68.808,174.290,22.838,153.902
C06264=1079.909,122.812,-68.827,174.292,22.841,153.902
C06265=1079.915,123.061,-68.847,174.293,22.842,153.902
C06266=1079.921,123.310,-68.866,174.296,22.845,153.903
C06267=1079.926,123.559,-68.885,174.297,22.847,153.903
C06268=1079.932,123.808,-68.905,174.299,22.849,153.903
C06269=1079.938,124.057,-68.924,174.301,22.851,153.903
C06270=1079.943,124.306,-68.945,174.303,22.854,153.903
C06271=1079.949,124.556,-68.964,174.304,22.856,153.904
C06272=1079.954,124.805,-68.984,174.306,22.858,153.904
C06273=1079.960,125.054,-69.003,174.308,22.860,153.904
C06274=1079.966,125.303,-69.023,174.310,22.862,153.904
C06275=1079.972,125.552,-69.043,174.311,22.865,153.904
C06276=1079.978,125.802,-69.062,174.314,22.867,153.905
C06277=1079.984,126.051,-69.081,174.316,22.869,153.905
C06278=1079.989,126.300,-69.102,174.318,22.871,153.905
C06279=1079.994,126.550,-69.121,174.320,22.873,153.905
C06280=1080.000,126.798,-69.141,174.321,22.876,153.905
C06281=1080.007,127.078,-69.163,174.323,22.878,153.905
C06282=1080.013,127.359,-69.185,174.326,22.881,153.906
C06283=1080.019,127.639,-69.207,174.328,22.883,153.906
C06284=1080.026,127.920,-69.229,174.330,22.886,153.906
C06285=1080.032,128.169,-69.249,174.331,22.888,153.906
C06286=1080.037,128.419,-69.268,174.334,22.890,153.906
C06287=1080.043,128.667,-69.288,174.335,22.892,153.907
C06288=1080.049,128.916,-69.308,174.338,22.894,153.907
C06289=1080.054,129.166,-69.328,174.339,22.896,153.907
C06290=1080.060,129.415,-69.348,174.341,22.899,153.907
C06291=1080.066,129.664,-69.367,174.343,22.901,153.907
C06292=1080.072,129.913,-69.387,174.345,22.903,153.907
C06293=1080.078,130.162,-69.407,174.347,22.905,153.908
C06294=1080.083,130.412,-69.427,174.349,22.907,153.908
C06295=1080.089,130.660,-69.447,174.351,22.910,153.908
C06296=1080.095,130.910,-69.466,174.352,22.911,153.908
C06297=1080.101,131.159,-69.486,174.355,22.914,153.908
C06298=1080.107,131.407,-69.506,174.357,22.917,153.908
C06299=1080.112,131.657,-69.526,174.358,22.918,153.909
C06300=1080.118,131.906,-69.546,174.361,22.921,153.909
C06301=1080.124,132.155,-69.566,174.362,22.923,153.909
C06302=1080.129,132.404,-69.585,174.364,22.925,153.909
C06303=1080.135,132.653,-69.606,174.366,22.927,153.909
C06304=1080.141,132.902,-69.626,174.368,22.930,153.909
C06305=1080.146,133.152,-69.646,174.370,22.932,153.910
C06306=1080.152,133.401,-69.666,174.372,22.934,153.910
C06307=1080.157,133.650,-69.686,174.374,22.936,153.910
C06308=1080.162,133.899,-69.705,174.375,22.938,153.910
C06309=1080.168,134.148,-69.725,174.378,22.941,153.910
C06310=1080.174,134.397,-69.746,174.380,22.943,153.911
C06311=1080.180,134.646,-69.766,174.381,22.945,153.911
C06312=1080.185,134.896,-69.786,174.384,22.947,153.911
C06313=1080.191,135.145,-69.806,174.385,22.949,153.911
C06314=1080.197,135.394,-69.827,174.387,22.952,153.911
C06315=1080.202,135.643,-69.846,174.390,22.954,153.911
C06316=1080.208,135.892,-69.867,174.391,22.956,153.912
C06317=1080.214,136.141,-69.887,174.393,22.958,153.912
C06318=1080.219,136.391,-69.907,174.395,22.960,153.912
C06319=1080.225,136.640,-69.927,174.397,22.963,153.912
C06320=1080.230,136.889,-69.947,174.399,22.965,153.912
C06321=1080.236,137.138,-69.967,174.401,22.967,153.912
C06322=1080.242,137.386,-69.987,174.403,22.969,153.913
C06323=1080.247,137.636,-70.008,174.405,22.971,153.913
C06324=1080.254,137.885,-70.028,174.407,22.973,153.913
C06325=1080.259,138.135,-70.048,174.409,22.976,153.913
C06326=1080.265,138.384,-70.068,174.410,22.978,153.913
C06327=1080.270,138.633,-70.088,174.413,22.980,153.913
C06328=1080.275,138.882,-70.109,174.414,22.982,153.914
C06329=1080.281,139.131,-70.129,174.417,22.984,153.914
C06330=1080.286,139.380,-70.150,174.419,22.987,153.914
C06331=1080.292,139.629,-70.170,174.420,22.989,153.914
C06332=1080.298,139.878,-70.190,174.423,22.991,153.914
C06333=1080.304,140.127,-70.210,174.424,22.993,153.914
C06334=1080.310,140.376,-70.231,174.426,22.995,153.915
C06335=1080.315,140.626,-70.252,174.429,22.998,153.915
C06336=1080.321,140.874,-70.271,174.430,23.000,153.915
C06337=1080.326,141.123,-70.292,174.432,23.002,153.915
C06338=1080.331,141.373,-70.313,174.435,23.004,153.915
C06339=1080.338,141.622,-70.333,174.436,23.006,153.915
C06340=1080.343,141.871,-70.353,174.438,23.009,153.916
C06341=1080.348,142.120,-70.374,174.440,23.011,153.916
C06342=1080.354,142.369,-70.394,174.442,23.013,153.916
C06343=1080.360,142.618,-70.415,174.444,23.015,153.916
C06344=1080.365,142.867,-70.435,174.446,23.017,153.916
C06345=1080.372,143.147,-70.458,174.448,23.019,153.916
C06346=1080.378,143.428,-70.481,174.450,23.022,153.917
C06347=1080.384,143.708,-70.504,174.453,23.024,153.917
C06348=1080.391,143.988,-70.528,174.455,23.027,153.917
C06349=1080.396,144.237,-70.548,174.457,23.029,153.917
C06350=1080.402,144.487,-70.569,174.459,23.032,153.917
C06351=1080.408,144.736,-70.589,174.461,23.034,153.918
C06352=1080.413,144.985,-70.610,174.463,23.036,153.918
C06353=1080.418,145.234,-70.630,174.466,23.038,153.918
C06354=1080.425,145.482,-70.651,174.467,23.040,153.918
C06355=1080.430,145.732,-70.672,174.469,23.042,153.918
C06356=1080.436,145.981,-70.692,174.471,23.044,153.918
C06357=1080.441,146.230,-70.713,174.473,23.046,153.918
C06358=1080.447,146.479,-70.733,174.475,23.049,153.919
C06359=1080.453,146.728,-70.755,174.477,23.051,153.919
C06360=1080.458,146.977,-70.775,174.479,23.053,153.919
C06361=1080.464,147.227,-70.796,174.481,23.056,153.919
C06362=1080.470,147.475,-70.816,174.483,23.057,153.919
C06363=1080.476,147.725,-70.837,174.485,23.060,153.919
C06364=1080.481,147.974,-70.858,174.488,23.062,153.920
C06365=1080.486,148.223,-70.878,174.489,23.064,153.920
C06366=1080.493,148.472,-70.899,174.491,23.066,153.920
C06367=1080.498,148.721,-70.920,174.494,23.068,153.920
C06368=1080.504,148.970,-70.941,174.495,23.070,153.920
C06369=1080.509,149.219,-70.961,174.497,23.072,153.920
C06370=1080.515,149.468,-70.983,174.500,23.075,153.921
C06371=1080.520,149.717,-71.003,174.501,23.077,153.921
C06372=1080.526,149.967,-71.024,174.504,23.079,153.921
C06373=1080.531,150.215,-71.045,174.506,23.081,153.921
C06374=1080.537,150.465,-71.066,174.507,23.083,153.921
C06375=1080.543,150.713,-71.087,174.510,23.085,153.921
C06376=1080.549,150.962,-71.107,174.512,23.088,153.922
C06377=1080.554,151.212,-71.128,174.514,23.090,153.922
C06378=1080.560,151.461,-71.149,174.516,23.092,153.922
C06379=1080.565,151.710,-71.170,174.518,23.094,153.922
C06380=1080.571,151.958,-71.191,174.520,23.097,153.922
C06381=1080.577,152.208,-71.212,174.522,23.099,153.922
C06382=1080.582,152.457,-71.233,174.524,23.101,153.922
C06383=1080.587,152.706,-71.254,174.526,23.103,153.923
C06384=1080.593,152.955,-71.275,174.528,23.105,153.923
C06385=1080.599,153.204,-71.296,174.530,23.107,153.923
C06386=1080.604,153.453,-71.317,174.533,23.109,153.923
C06387=1080.610,153.702,-71.338,174.534,23.111,153.923
C06388=1080.616,153.951,-71.359,174.536,23.114,153.923
C06389=1080.621,154.200,-71.380,174.539,23.116,153.923
C06390=1080.627,154.450,-71.401,174.541,23.118,153.924
C06391=1080.633,154.698,-71.422,174.542,23.120,153.924
C06392=1080.638,154.947,-71.444,174.545,23.122,153.924
C06393=1080.644,155.197,-71.465,174.547,23.124,153.924
C06394=1080.650,155.445,-71.486,174.549,23.126,153.924
C06395=1080.655,155.695,-71.507,174.551,23.129,153.924
C06396=1080.661,155.943,-71.528,174.553,23.131,153.925
C06397=1080.665,156.193,-71.549,174.556,23.133,153.925
C06398=1080.672,156.442,-71.571,174.557,23.135,153.925
C06399=1080.677,156.691,-71.592,174.559,23.137,153.925
C06400=1080.682,156.940,-71.613,174.562,23.140,153.925
C06401=1080.689,157.189,-71.634,174.563,23.141,153.925
C06402=1080.694,157.437,-71.656,174.565,23.144,153.925
C06403=1080.700,157.687,-71.676,174.568,23.146,153.926
C06404=1080.706,157.936,-71.698,174.570,23.148,153.926
C06405=1080.710,158.185,-71.720,174.572,23.150,153.926
C06406=1080.716,158.434,-71.741,174.574,23.152,153.926
C06407=1080.722,158.683,-71.762,174.576,23.155,153.926
C06408=1080.728,158.932,-71.783,174.579,23.157,153.926
C06409=1080.734,159.212,-71.807,174.581,23.160,153.927
C06410=1080.740,159.492,-71.831,174.583,23.162,153.927
C06411=1080.747,159.772,-71.855,174.585,23.164,153.927
C06412=1080.753,160.052,-71.879,174.588,23.166,153.927
C06413=1080.759,160.301,-71.900,174.590,23.169,153.927
C06414=1080.765,160.550,-71.922,174.592,23.170,153.927
C06415=1080.770,160.799,-71.944,174.594,23.173,153.927
C06416=1080.775,161.049,-71.964,174.596,23.175,153.928
C06417=1080.781,161.298,-71.986,174.599,23.177,153.928
C06418=1080.787,161.546,-72.007,174.600,23.179,153.928
C06419=1080.792,161.795,-72.029,174.602,23.181,153.928
C06420=1080.798,162.044,-72.051,174.605,23.184,153.928
C06421=1080.802,162.294,-72.072,174.607,23.186,153.928
C06422=1080.809,162.543,-72.094,174.609,23.188,153.928
C06423=1080.814,162.791,-72.115,174.611,23.190,153.929
C06424=1080.819,163.040,-72.137,174.613,23.193,153.929
C06425=1080.825,163.289,-72.158,174.615,23.195,153.929
C06426=1080.830,163.538,-72.180,174.617,23.197,153.929
C06427=1080.836,163.787,-72.202,174.619,23.199,153.929
C06428=1080.841,164.036,-72.224,174.622,23.201,153.929
C06429=1080.847,164.285,-72.245,174.624,23.204,153.930
C06430=1080.852,164.534,-72.267,174.626,23.206,153.930
C06431=1080.857,164.783,-72.288,174.628,23.208,153.930
C06432=1080.863,165.033,-72.310,174.630,23.210,153.930
C06433=1080.868,165.281,-72.331,174.632,23.212,153.930
C06434=1080.874,165.531,-72.354,174.635,23.214,153.930
C06435=1080.879,165.779,-72.375,174.636,23.216,153.931
C06436=1080.885,166.029,-72.397,174.639,23.219,153.931
C06437=1080.890,166.277,-72.418,174.641,23.221,153.931
C06438=1080.896,166.527,-72.441,174.643,23.223,153.931
C06439=1080.901,166.775,-72.462,174.645,23.226,153.931
C06440=1080.907,167.025,-72.484,174.647,23.228,153.931
C06441=1080.912,167.273,-72.506,174.649,23.230,153.932
C06442=1080.918,167.522,-72.528,174.652,23.232,153.932
C06443=1080.923,167.771,-72.550,174.654,23.234,153.932
C06444=1080.929,168.020,-72.572,174.656,23.237,153.932
C06445=1080.934,168.269,-72.593,174.658,23.239,153.932
C06446=1080.940,168.518,-72.615,174.660,23.241,153.932
C06447=1080.945,168.767,-72.637,174.662,23.243,153.932
C06448=1080.951,169.016,-72.659,174.665,23.245,153.933
C06449=1080.956,169.265,-72.680,174.667,23.248,153.933
C06450=1080.962,169.514,-72.702,174.669,23.249,153.933
C06451=1080.967,169.763,-72.725,174.671,23.252,153.933
C06452=1080.973,170.012,-72.746,174.673,23.254,153.933
C06453=1080.979,170.261,-72.769,174.676,23.256,153.933
C06454=1080.984,170.510,-72.790,174.678,23.258,153.933
C06455=1080.990,170.759,-72.812,174.680,23.260,153.933
C06456=1080.995,171.008,-72.833,174.682,23.262,153.934
C06457=1081.001,171.257,-72.856,174.684,23.264,153.934
C06458=1081.006,171.506,-72.879,174.687,23.267,153.934
C06459=1081.012,171.755,-72.900,174.689,23.269,153.934
C06460=1081.017,172.004,-72.922,174.691,23.271,153.934
C06461=1081.023,172.252,-72.944,174.693,23.273,153.934
C06462=1081.029,172.502,-72.966,174.695,23.275,153.935
C06463=1081.034,172.751,-72.989,174.697,23.277,153.935
C06464=1081.039,173.000,-73.010,174.700,23.280,153.935
C06465=1081.045,173.249,-73.033,174.702,23.282,153.935
C06466=1081.051,173.498,-73.054,174.705,23.284,153.935
C06467=1081.056,173.747,-73.076,174.706,23.286,153.935
C06468=1081.062,173.996,-73.099,174.708,23.288,153.935
C06469=1081.068,174.245,-73.121,174.711,23.290,153.936
C06470=1081.073,174.494,-73.143,174.713,23.292,153.936
C06471=1081.079,174.742,-73.166,174.716,23.294,153.936
C06472=1081.085,174.992,-73.187,174.718,23.297,153.936
C06473=1081.091,175.272,-73.212,174.720,23.299,153.936
C06474=1081.098,175.551,-73.238,174.723,23.301,153.936
C06475=1081.103,175.831,-73.263,174.725,23.304,153.936
C06476=1081.110,176.111,-73.287,174.727,23.306,153.937
C06477=1081.115,176.359,-73.310,174.729,23.308,153.937
C06478=1081.121,176.608,-73.331,174.732,23.310,153.937
C06479=1081.127,176.857,-73.354,174.734,23.312,153.937
C06480=1081.132,177.106,-73.376,174.737,23.315,153.937
C06481=1081.138,177.354,-73.398,174.739,23.317,153.937
C06482=1081.144,177.604,-73.421,174.741,23.319,153.937
C06483=1081.149,177.853,-73.443,174.743,23.321,153.937
C06484=1081.155,178.101,-73.465,174.745,23.323,153.938
C06485=1081.160,178.351,-73.487,174.748,23.325,153.938
C06486=1081.166,178.600,-73.510,174.750,23.327,153.938
C06487=1081.173,178.848,-73.532,174.752,23.329,153.938
C06488=1081.177,179.097,-73.554,174.755,23.332,153.938
C06489=1081.183,179.346,-73.577,174.757,23.334,153.938
C06490=1081.189,179.595,-73.599,174.760,23.336,153.938
C06491=1081.195,179.844,-73.622,174.761,23.338,153.938
C06492=1081.201,180.094,-73.644,174.764,23.340,153.938
C06493=1081.206,180.342,-73.667,174.766,23.342,153.939
C06494=1081.212,180.590,-73.689,174.768,23.344,153.939
C06495=1081.218,180.840,-73.711,174.771,23.347,153.939
C06496=1081.223,181.089,-73.734,174.773,23.348,153.939
C06497=1081.229,181.338,-73.756,174.775,23.351,153.939
C06498=1081.235,181.587,-73.779,174.778,23.353,153.939
C06499=1081.240,181.835,-73.801,174.780,23.355,153.939
C06500=1081.246,182.085,-73.824,174.782,23.357,153.940
C06501=1081.251,182.333,-73.846,174.784,23.359,153.940
C06502=1081.258,182.582,-73.869,174.786,23.361,153.940
C06503=1081.263,182.832,-73.891,174.789,23.363,153.940
C06504=1081.269,183.080,-73.914,174.791,23.365,153.940
C06505=1081.275,183.329,-73.937,174.794,23.367,153.940
C06506=1081.281,183.578,-73.959,174.796,23.369,153.940
C06507=1081.286,183.827,-73.981,174.798,23.371,153.940
C06508=1081.292,184.076,-74.004,174.801,23.374,153.940
C06509=1081.298,184.325,-74.027,174.803,23.375,153.940
C06510=1081.304,184.573,-74.049,174.806,23.378,153.941
C06511=1081.309,184.823,-74.072,174.807,23.380,153.941
C06512=1081.315,185.072,-74.095,174.809,23.382,153.941
C06513=1081.321,185.320,-74.118,174.812,23.384,153.941
C06514=1081.326,185.569,-74.140,174.814,23.386,153.941
C06515=1081.331,185.818,-74.164,174.817,23.389,153.941
C06516=1081.337,186.067,-74.187,174.819,23.391,153.941
C06517=1081.342,186.316,-74.209,174.821,23.393,153.942
C06518=1081.348,186.565,-74.232,174.824,23.395,153.942
C06519=1081.353,186.813,-74.254,174.826,23.397,153.942
C06520=1081.359,187.062,-74.277,174.828,23.400,153.942
C06521=1081.364,187.311,-74.301,174.831,23.402,153.942
C06522=1081.369,187.560,-74.324,174.833,23.404,153.942
C06523=1081.375,187.809,-74.347,174.835,23.406,153.942
C06524=1081.381,188.058,-74.370,174.838,23.408,153.942
C06525=1081.386,188.306,-74.392,174.840,23.410,153.943
C06526=1081.392,188.555,-74.415,174.843,23.413,153.943
C06527=1081.397,188.804,-74.439,174.844,23.414,153.943
C06528=1081.402,189.054,-74.461,174.846,23.417,153.943
C06529=1081.408,189.303,-74.484,174.849,23.419,153.943
C06530=1081.414,189.552,-74.507,174.851,23.421,153.943
C06531=1081.419,189.801,-74.530,174.854,23.423,153.944
C06532=1081.424,190.050,-74.553,174.856,23.426,153.944
C06533=1081.430,190.298,-74.576,174.858,23.428,153.944
C06534=1081.436,190.546,-74.600,174.861,23.430,153.944
C06535=1081.441,190.795,-74.623,174.863,23.432,153.944
C06536=1081.447,191.044,-74.645,174.865,23.435,153.944
C06537=1081.452,191.324,-74.672,174.868,23.437,153.944
C06538=1081.459,191.603,-74.698,174.871,23.440,153.944
C06539=1081.465,191.883,-74.723,174.873,23.442,153.945
C06540=1081.471,192.162,-74.749,174.876,23.444,153.945
C06541=1081.477,192.410,-74.773,174.878,23.446,153.945
C06542=1081.483,192.659,-74.796,174.880,23.448,153.945
C06543=1081.488,192.908,-74.819,174.883,23.451,153.945
C06544=1081.493,193.157,-74.842,174.885,23.453,153.945
C06545=1081.499,193.406,-74.865,174.888,23.455,153.945
C06546=1081.505,193.655,-74.888,174.890,23.457,153.946
C06547=1081.511,193.904,-74.911,174.892,23.460,153.946
C06548=1081.516,194.153,-74.935,174.895,23.461,153.946
C06549=1081.522,194.401,-74.958,174.897,23.464,153.946
C06550=1081.527,194.650,-74.981,174.899,23.466,153.946
C06551=1081.532,194.900,-75.005,174.902,23.468,153.946
C06552=1081.538,195.148,-75.028,174.904,23.470,153.946
C06553=1081.544,195.397,-75.051,174.907,23.473,153.947
C06554=1081.550,195.646,-75.074,174.909,23.475,153.947
C06555=1081.555,195.895,-75.098,174.911,23.477,153.947
C06556=1081.561,196.143,-75.121,174.914,23.479,153.947
C06557=1081.567,196.392,-75.144,174.916,23.481,153.947
C06558=1081.572,196.641,-75.168,174.919,23.483,153.947
C06559=1081.578,196.890,-75.192,174.921,23.485,153.947
C06560=1081.584,197.139,-75.215,174.923,23.488,153.947
C06561=1081.589,197.388,-75.238,174.927,23.490,153.948
C06562=1081.595,197.637,-75.262,174.929,23.493,153.948
C06563=1081.601,197.885,-75.285,174.931,23.494,153.948
C06564=1081.606,198.135,-75.309,174.934,23.496,153.948
C06565=1081.612,198.383,-75.332,174.936,23.499,153.948
C06566=1081.617,198.632,-75.355,174.939,23.501,153.948
C06567=1081.622,198.881,-75.379,174.941,23.503,153.948
C06568=1081.629,199.129,-75.402,174.943,23.505,153.948
C06569=1081.634,199.378,-75.425,174.946,23.507,153.948
C06570=1081.640,199.628,-75.450,174.948,23.509,153.949
C06571=1081.646,199.876,-75.473,174.951,23.512,153.949
C06572=1081.651,200.125,-75.497,174.953,23.514,153.949
C06573=1081.657,200.374,-75.520,174.955,23.516,153.949
C06574=1081.663,200.622,-75.544,174.958,23.518,153.949
C06575=1081.668,200.871,-75.567,174.960,23.520,153.949
C06576=1081.674,201.120,-75.591,174.963,23.522,153.949
C06577=1081.680,201.369,-75.614,174.965,23.524,153.949
C06578=1081.686,201.618,-75.639,174.967,23.527,153.950
C06579=1081.691,201.867,-75.662,174.970,23.529,153.950
C06580=1081.697,202.115,-75.686,174.972,23.531,153.950
C06581=1081.702,202.364,-75.709,174.975,23.533,153.950
C06582=1081.709,202.613,-75.733,174.977,23.535,153.950
C06583=1081.714,202.862,-75.756,174.980,23.538,153.950
C06584=1081.719,203.111,-75.781,174.983,23.540,153.950
C06585=1081.725,203.359,-75.804,174.985,23.542,153.950
C06586=1081.730,203.609,-75.828,174.987,23.544,153.951
C06587=1081.736,203.857,-75.852,174.990,23.547,153.951
C06588=1081.742,204.105,-75.876,174.992,23.549,153.951
C06589=1081.747,204.355,-75.900,174.995,23.551,153.951
C06590=1081.753,204.604,-75.923,174.997,23.553,153.951
C06591=1081.759,204.852,-75.947,174.999,23.555,153.951
C06592=1081.764,205.101,-75.971,175.002,23.557,153.951
C06593=1081.770,205.350,-75.995,175.004,23.560,153.952
C06594=1081.775,205.598,-76.019,175.006,23.562,153.952
C06595=1081.781,205.848,-76.043,175.010,23.564,153.952
C06596=1081.787,206.096,-76.067,175.012,23.567,153.952
C06597=1081.792,206.345,-76.091,175.014,23.569,153.952
C06598=1081.797,206.594,-76.115,175.017,23.571,153.952
C06599=1081.803,206.842,-76.138,175.019,23.573,153.952
C06600=1081.809,207.092,-76.163,175.021,23.576,153.952
C06601=1081.832,208.124,-76.262,175.116,23.626,153.950
C06602=1081.841,208.519,-76.301,175.120,23.630,153.951
C06603=1081.850,208.914,-76.340,175.124,23.635,153.951
C06604=1081.859,209.311,-76.379,175.127,23.640,153.952
C06605=1081.868,209.706,-76.419,175.131,23.646,153.953
C06606=1081.874,209.955,-76.443,175.134,23.649,153.953
C06607=1081.879,210.204,-76.468,175.136,23.652,153.953
C06608=1081.885,210.453,-76.492,175.138,23.655,153.954
C06609=1081.891,210.701,-76.517,175.140,23.658,153.954
C06610=1081.896,210.950,-76.541,175.143,23.662,153.954
C06611=1081.902,211.199,-76.566,175.145,23.664,153.955
C06612=1081.907,211.447,-76.591,175.147,23.668,153.955
C06613=1081.913,211.696,-76.616,175.150,23.671,153.955
C06614=1081.919,211.945,-76.640,175.152,23.674,153.956
C06615=1081.925,212.194,-76.665,175.154,23.677,153.956
C06616=1081.930,212.442,-76.689,175.157,23.680,153.956
C06617=1081.936,212.691,-76.715,175.160,23.684,153.957
C06618=1081.942,212.939,-76.739,175.162,23.687,153.957
C06619=1081.948,213.189,-76.764,175.164,23.690,153.957
C06620=1081.953,213.437,-76.789,175.167,23.693,153.958
C06621=1081.959,213.686,-76.813,175.169,23.696,153.958
C06622=1081.964,213.934,-76.839,175.171,23.699,153.958
C06623=1081.970,214.183,-76.863,175.174,23.703,153.959
C06624=1081.975,214.431,-76.888,175.176,23.706,153.959
C06625=1081.981,214.681,-76.913,175.178,23.709,153.960
C06626=1081.987,214.929,-76.938,175.180,23.712,153.960
C06627=1081.992,215.178,-76.963,175.183,23.716,153.960
C06628=1081.998,215.427,-76.989,175.186,23.718,153.961
C06629=1082.004,215.676,-77.013,175.188,23.722,153.961
C06630=1082.010,215.924,-77.038,175.191,23.725,153.961
C06631=1082.015,216.173,-77.062,175.193,23.728,153.962
C06632=1082.021,216.422,-77.088,175.195,23.731,153.962
C06633=1082.026,216.670,-77.113,175.198,23.734,153.962
C06634=1082.032,216.919,-77.138,175.200,23.738,153.963
C06635=1082.038,217.167,-77.163,175.202,23.741,153.963
C06636=1082.043,217.417,-77.188,175.205,23.744,153.963
C06637=1082.049,217.665,-77.213,175.207,23.747,153.964
C06638=1082.055,217.913,-77.238,175.209,23.750,153.964
C06639=1082.061,218.163,-77.263,175.212,23.754,153.964
C06640=1082.065,218.411,-77.289,175.214,23.757,153.965
C06641=1082.072,218.659,-77.314,175.217,23.759,153.965
C06642=1082.078,218.909,-77.339,175.220,23.763,153.966
C06643=1082.083,219.157,-77.364,175.222,23.766,153.966
C06644=1082.089,219.406,-77.389,175.224,23.769,153.966
C06645=1082.094,219.655,-77.414,175.227,23.773,153.967
C06646=1082.100,219.903,-77.439,175.229,23.775,153.967
C06647=1082.106,220.152,-77.465,175.231,23.779,153.967
C06648=1082.112,220.401,-77.490,175.234,23.782,153.968
C06649=1082.117,220.649,-77.515,175.236,23.785,153.968
C06650=1082.123,220.898,-77.541,175.238,23.788,153.968
C06651=1082.129,221.147,-77.566,175.241,23.791,153.969
C06652=1082.134,221.395,-77.591,175.243,23.795,153.969
C06653=1082.141,221.643,-77.616,175.246,23.797,153.969
C06654=1082.149,222.043,-77.657,175.250,23.803,153.970
C06655=1082.158,222.443,-77.698,175.254,23.808,153.971
C06656=1082.167,222.843,-77.739,175.258,23.813,153.971
C06657=1082.177,223.243,-77.780,175.262,23.818,153.972
C06658=1082.182,223.492,-77.805,175.264,23.822,153.972
C06659=1082.187,223.740,-77.831,175.267,23.825,153.972
C06660=1082.193,223.989,-77.856,175.269,23.828,153.973
C06661=1082.199,224.238,-77.882,175.271,23.831,153.973
C06662=1082.205,224.486,-77.907,175.274,23.834,153.973
C06663=1082.210,224.735,-77.933,175.276,23.837,153.974
C06664=1082.216,224.984,-77.958,175.279,23.841,153.974
C06665=1082.222,225.233,-77.984,175.281,23.844,153.975
C06666=1082.227,225.481,-78.010,175.283,23.847,153.975
C06667=1082.233,225.730,-78.035,175.286,23.850,153.975
C06668=1082.238,225.978,-78.061,175.289,23.853,153.976
C06669=1082.244,226.227,-78.086,175.291,23.857,153.976
C06670=1082.250,226.475,-78.112,175.294,23.860,153.976
C06671=1082.256,226.723,-78.138,175.296,23.863,153.977
C06672=1082.261,226.972,-78.164,175.299,23.867,153.977
C06673=1082.268,227.221,-78.189,175.301,23.869,153.977
C06674=1082.273,227.470,-78.215,175.303,23.873,153.978
C06675=1082.278,227.718,-78.241,175.306,23.876,153.978
C06676=1082.284,227.967,-78.266,175.308,23.879,153.978
C06677=1082.290,228.216,-78.292,175.310,23.882,153.979
C06678=1082.296,228.464,-78.318,175.313,23.885,153.979
C06679=1082.301,228.713,-78.344,175.315,23.888,153.979
C06680=1082.306,228.961,-78.369,175.319,23.892,153.980
C06681=1082.313,229.210,-78.395,175.321,23.895,153.980
C06682=1082.318,229.459,-78.421,175.323,23.898,153.981
C06683=1082.325,229.707,-78.447,175.326,23.901,153.981
C06684=1082.330,229.956,-78.473,175.328,23.904,153.981
C06685=1082.335,230.205,-78.499,175.331,23.907,153.981
C06686=1082.342,230.453,-78.525,175.333,23.911,153.982
C06687=1082.347,230.701,-78.550,175.335,23.914,153.982
C06688=1082.352,230.950,-78.576,175.338,23.917,153.983
C06689=1082.358,231.199,-78.602,175.340,23.920,153.983
C06690=1082.364,231.448,-78.629,175.343,23.924,153.983
C06691=1082.370,231.696,-78.654,175.346,23.926,153.984
C06692=1082.375,231.945,-78.680,175.349,23.930,153.984
C06693=1082.381,232.194,-78.707,175.351,23.933,153.984
C06694=1082.386,232.443,-78.733,175.353,23.936,153.985
C06695=1082.392,232.690,-78.759,175.356,23.940,153.985
C06696=1082.398,232.939,-78.784,175.358,23.943,153.986
C06697=1082.403,233.188,-78.810,175.361,23.946,153.986
C06698=1082.409,233.436,-78.837,175.363,23.949,153.986
C06699=1082.415,233.685,-78.863,175.366,23.953,153.987
C06700=1082.420,233.934,-78.889,175.368,23.956,153.987
C06701=1082.426,234.183,-78.915,175.370,23.959,153.987
C06702=1082.432,234.431,-78.942,175.373,23.962,153.988
C06703=1082.438,234.680,-78.967,175.376,23.965,153.988
C06704=1082.444,234.928,-78.994,175.379,23.969,153.988
C06705=1082.448,235.176,-79.019,175.381,23.972,153.989
C06706=1082.457,235.568,-79.061,175.385,23.977,153.989
C06707=1082.466,235.959,-79.102,175.389,23.982,153.990
C06708=1082.475,236.350,-79.144,175.392,23.987,153.990
C06709=1082.484,236.741,-79.186,175.397,23.992,153.991
C06710=1082.489,236.990,-79.212,175.399,23.995,153.991
C06711=1082.495,237.239,-79.238,175.402,23.999,153.992
C06712=1082.502,237.487,-79.265,175.404,24.002,153.992
C06713=1082.507,237.736,-79.290,175.407,24.005,153.992
C06714=1082.513,237.984,-79.317,175.409,24.008,153.993
C06715=1082.519,238.232,-79.344,175.412,24.011,153.993
C06716=1082.524,238.481,-79.370,175.415,24.014,153.993
C06717=1082.530,238.730,-79.396,175.417,24.018,153.994
C06718=1082.536,238.978,-79.423,175.420,24.021,153.994
C06719=1082.541,239.227,-79.449,175.422,24.024,153.995
C06720=1082.547,239.475,-79.476,175.425,24.027,153.995
C06721=1082.553,239.724,-79.502,175.427,24.031,153.995
C06722=1082.558,239.973,-79.530,175.430,24.034,153.996
C06723=1082.564,240.221,-79.556,175.432,24.037,153.996
C06724=1082.569,240.470,-79.582,175.435,24.041,153.996
C06725=1082.575,240.719,-79.609,175.437,24.043,153.997
C06726=1082.581,240.967,-79.636,175.440,24.047,153.997
C06727=1082.587,241.215,-79.662,175.443,24.050,153.997
C06728=1082.593,241.464,-79.689,175.446,24.053,153.998
C06729=1082.598,241.712,-79.716,175.448,24.056,153.998
C06730=1082.604,241.961,-79.742,175.451,24.060,153.999
C06731=1082.610,242.210,-79.768,175.453,24.063,153.999
C06732=1082.615,242.458,-79.795,175.455,24.066,153.999
C06733=1082.621,242.706,-79.822,175.458,24.069,153.999
C06734=1082.627,242.956,-79.849,175.460,24.072,154.000
C06735=1082.633,243.204,-79.876,175.463,24.076,154.000
C06736=1082.638,243.452,-79.902,175.465,24.079,154.001
C06737=1082.644,243.701,-79.929,175.469,24.082,154.001
C06738=1082.649,243.949,-79.956,175.471,24.085,154.001
C06739=1082.655,244.198,-79.983,175.474,24.089,154.002
C06740=1082.661,244.446,-80.010,175.476,24.092,154.002
C06741=1082.666,244.694,-80.036,175.479,24.095,154.002
C06742=1082.671,244.943,-80.064,175.481,24.098,154.003
C06743=1082.677,245.191,-80.090,175.484,24.102,154.003
C06744=1082.684,245.441,-80.117,175.486,24.105,154.004
C06745=1082.689,245.689,-80.144,175.489,24.108,154.004
C06746=1082.694,245.938,-80.171,175.491,24.111,154.004
C06747=1082.700,246.186,-80.198,175.494,24.115,154.005
C06748=1082.706,246.434,-80.226,175.496,24.118,154.005
C06749=1082.711,246.682,-80.252,175.499,24.121,154.005
C06750=1082.718,246.931,-80.279,175.502,24.124,154.006
C06751=1082.723,247.180,-80.306,175.505,24.128,154.006
C06752=1082.728,247.428,-80.333,175.508,24.131,154.006
C06753=1082.734,247.677,-80.360,175.510,24.134,154.007
C06754=1082.740,247.925,-80.388,175.513,24.138,154.007
C06755=1082.745,248.173,-80.414,175.515,24.141,154.008
C06756=1082.750,248.422,-80.442,175.518,24.145,154.008
C06757=1082.757,248.671,-80.469,175.520,24.147,154.008
C06758=1082.765,249.055,-80.511,175.525,24.153,154.009
C06759=1082.773,249.440,-80.553,175.528,24.158,154.010
C06760=1082.782,249.824,-80.596,175.533,24.163,154.010
C06761=1082.791,250.208,-80.638,175.536,24.168,154.011
C06762=1082.797,250.457,-80.665,175.539,24.172,154.011
C06763=1082.802,250.706,-80.692,175.541,24.175,154.012
C06764=1082.808,250.953,-80.720,175.545,24.178,154.012
C06765=1082.813,251.202,-80.747,175.547,24.181,154.012
C06766=1082.819,251.451,-80.774,175.550,24.185,154.013
C06767=1082.825,251.699,-80.802,175.552,24.188,154.013
C06768=1082.830,251.948,-80.829,175.555,24.192,154.013
C06769=1082.836,252.195,-80.856,175.557,24.194,154.014
C06770=1082.841,252.445,-80.884,175.560,24.198,154.014
C06771=1082.847,252.693,-80.911,175.562,24.201,154.015
C06772=1082.853,252.941,-80.939,175.565,24.205,154.015
C06773=1082.859,253.189,-80.966,175.568,24.208,154.015
C06774=1082.864,253.438,-80.994,175.570,24.211,154.016
C06775=1082.870,253.686,-81.021,175.573,24.214,154.016
C06776=1082.875,253.935,-81.048,175.575,24.218,154.016
C06777=1082.881,254.183,-81.076,175.578,24.221,154.017
C06778=1082.887,254.432,-81.103,175.581,24.224,154.017
C06779=1082.892,254.680,-81.131,175.584,24.227,154.017
C06780=1082.898,254.929,-81.159,175.586,24.231,154.018
C06781=1082.904,255.177,-81.186,175.589,24.234,154.018
C06782=1082.909,255.425,-81.214,175.592,24.238,154.019
C06783=1082.915,255.674,-81.242,175.594,24.240,154.019
C06784=1082.921,255.922,-81.269,175.597,24.244,154.019
C06785=1082.926,256.171,-81.296,175.599,24.247,154.020
C06786=1082.932,256.420,-81.325,175.602,24.251,154.020
C06787=1082.938,256.667,-81.352,175.604,24.254,154.020
C06788=1082.944,256.916,-81.380,175.607,24.257,154.021
C06789=1082.949,257.165,-81.407,175.611,24.261,154.021
C06790=1082.955,257.413,-81.435,175.613,24.264,154.022
C06791=1082.961,257.661,-81.463,175.616,24.267,154.022
C06792=1082.966,257.910,-81.490,175.618,24.270,154.022
C06793=1082.973,258.158,-81.518,175.621,24.274,154.023
C06794=1082.978,258.406,-81.546,175.624,24.277,154.023
C06795=1082.984,258.654,-81.574,175.626,24.280,154.023
C06796=1082.990,258.903,-81.602,175.629,24.283,154.024
C06797=1082.995,259.152,-81.629,175.631,24.287,154.024
C06798=1083.001,259.400,-81.657,175.634,24.290,154.025
C06799=1083.007,259.648,-81.685,175.637,24.293,154.025
C06800=1083.013,259.897,-81.713,175.640,24.296,154.025
C06801=1083.019,260.145,-81.741,175.643,24.300,154.026
C06802=1083.025,260.394,-81.769,175.645,24.303,154.026
C06803=1083.031,260.641,-81.797,175.648,24.306,154.026
C06804=1083.036,260.891,-81.824,175.651,24.310,154.027
C06805=1083.042,261.139,-81.852,175.653,24.313,154.027
C06806=1083.048,261.388,-81.881,175.656,24.317,154.028
C06807=1083.054,261.635,-81.908,175.658,24.319,154.028
C06808=1083.060,261.884,-81.936,175.661,24.323,154.028
C06809=1083.065,262.132,-81.964,175.664,24.326,154.029
C06810=1083.070,262.343,-81.988,175.667,24.329,154.029
C06811=1083.076,262.555,-82.012,175.669,24.332,154.029
C06812=1083.080,262.767,-82.036,175.671,24.334,154.029
C06813=1083.085,262.978,-82.060,175.673,24.337,154.030
C06814=1083.090,263.189,-82.084,175.675,24.340,154.030
C06815=1083.095,263.400,-82.107,175.678,24.343,154.030
C06816=1083.100,263.611,-82.131,175.680,24.346,154.031
C06817=1083.105,263.823,-82.155,175.682,24.348,154.031
C06818=1083.111,264.071,-82.183,175.685,24.352,154.031
C06819=1083.117,264.320,-82.212,175.688,24.355,154.032
C06820=1083.122,264.568,-82.240,175.690,24.359,154.032
C06821=1083.128,264.816,-82.269,175.694,24.362,154.033
C06822=1083.133,265.064,-82.297,175.696,24.365,154.033
C06823=1083.139,265.313,-82.325,175.699,24.368,154.033
C06824=1083.145,265.561,-82.353,175.702,24.372,154.034
C06825=1083.151,265.810,-82.381,175.704,24.375,154.034
C06826=1083.157,266.037,-82.408,175.707,24.379,154.035
C06827=1083.162,266.265,-82.434,175.709,24.381,154.035
C06828=1083.167,266.493,-82.459,175.711,24.385,154.035
C06829=1083.172,266.721,-82.485,175.714,24.388,154.036
C06830=1083.177,266.948,-82.511,175.717,24.391,154.036
C06831=1083.182,267.177,-82.538,175.719,24.394,154.036
C06832=1083.187,267.405,-82.564,175.722,24.397,154.037
C06833=1083.193,267.632,-82.590,175.724,24.400,154.037
C06834=1083.199,267.880,-82.618,175.727,24.404,154.037
C06835=1083.205,268.129,-82.646,175.729,24.407,154.038
C06836=1083.210,268.376,-82.675,175.732,24.410,154.038
C06837=1083.216,268.625,-82.703,175.735,24.413,154.039
C06838=1083.221,268.874,-82.732,175.737,24.417,154.039
C06839=1083.227,269.122,-82.761,175.740,24.420,154.039
C06840=1083.233,269.370,-82.789,175.743,24.424,154.040
C06841=1083.239,269.619,-82.818,175.746,24.427,154.040
C06842=1083.245,269.867,-82.846,175.749,24.430,154.041
C06843=1083.250,270.115,-82.875,175.752,24.434,154.041
C06844=1083.255,270.363,-82.904,175.754,24.437,154.041
C06845=1083.261,270.612,-82.932,175.757,24.441,154.042
C06846=1083.268,270.860,-82.961,175.760,24.444,154.042
C06847=1083.273,271.108,-82.989,175.762,24.447,154.043
C06848=1083.279,271.356,-83.018,175.765,24.451,154.043
C06849=1083.284,271.605,-83.047,175.768,24.455,154.043
C06850=1083.290,271.853,-83.076,175.770,24.457,154.044
C06851=1083.296,272.101,-83.104,175.773,24.461,154.044
C06852=1083.302,272.349,-83.133,175.776,24.464,154.044
C06853=1083.307,272.598,-83.162,175.779,24.468,154.045
C06854=1083.313,272.846,-83.191,175.782,24.471,154.045
C06855=1083.319,273.094,-83.220,175.785,24.475,154.046
C06856=1083.325,273.343,-83.249,175.788,24.478,154.046
C06857=1083.330,273.591,-83.277,175.790,24.481,154.047
C06858=1083.336,273.839,-83.306,175.793,24.485,154.047
C06859=1083.342,274.088,-83.335,175.796,24.488,154.047
C06860=1083.347,274.335,-83.364,175.798,24.492,154.048
C06861=1083.354,274.583,-83.393,175.801,24.495,154.048
C06862=1083.359,274.832,-83.422,175.804,24.499,154.049
C06863=1083.365,275.081,-83.451,175.806,24.502,154.049
C06864=1083.370,275.328,-83.480,175.809,24.505,154.049
C06865=1083.376,275.577,-83.509,175.812,24.509,154.050
C06866=1083.385,275.962,-83.554,175.817,24.515,154.050
C06867=1083.394,276.346,-83.599,175.820,24.520,154.051
C06868=1083.403,276.731,-83.644,175.825,24.525,154.052
C06869=1083.411,277.115,-83.689,175.829,24.530,154.052
C06870=1083.417,277.363,-83.718,175.832,24.534,154.053
C06871=1083.423,277.612,-83.748,175.834,24.537,154.053
C06872=1083.429,277.860,-83.777,175.837,24.541,154.054
C06873=1083.434,278.108,-83.805,175.840,24.544,154.054
C06874=1083.440,278.356,-83.835,175.844,24.548,154.054
C06875=1083.445,278.605,-83.864,175.846,24.551,154.055
C06876=1083.452,278.853,-83.893,175.849,24.555,154.055
C06877=1083.457,279.101,-83.923,175.852,24.558,154.056
C06878=1083.463,279.349,-83.952,175.854,24.561,154.056
C06879=1083.468,279.597,-83.981,175.857,24.565,154.056
C06880=1083.475,279.845,-84.010,175.860,24.568,154.057
C06881=1083.480,280.094,-84.040,175.863,24.572,154.057
C06882=1083.486,280.342,-84.069,175.865,24.575,154.058
C06883=1083.492,280.590,-84.098,175.868,24.579,154.058
C06884=1083.498,280.838,-84.128,175.871,24.583,154.059
C06885=1083.504,281.087,-84.157,175.874,24.586,154.059
C06886=1083.509,281.335,-84.187,175.876,24.589,154.059
C06887=1083.515,281.583,-84.215,175.879,24.593,154.060
C06888=1083.520,281.831,-84.245,175.882,24.596,154.060
C06889=1083.526,282.079,-84.275,175.885,24.600,154.061
C06890=1083.532,282.327,-84.305,175.887,24.604,154.061
C06891=1083.538,282.576,-84.334,175.890,24.607,154.062
C06892=1083.543,282.824,-84.364,175.893,24.611,154.062
C06893=1083.549,283.072,-84.393,175.897,24.614,154.062
C06894=1083.555,283.320,-84.422,175.899,24.617,154.063
C06895=1083.560,283.568,-84.452,175.902,24.621,154.063
C06896=1083.566,283.816,-84.482,175.905,24.625,154.064
C06897=1083.571,284.065,-84.512,175.908,24.628,154.064
C06898=1083.578,284.313,-84.541,175.911,24.632,154.064
C06899=1083.583,284.560,-84.571,175.913,24.635,154.065
C06900=1083.589,284.809,-84.601,175.916,24.639,154.065
C06901=1083.595,285.057,-84.630,175.919,24.643,154.066
C06902=1083.601,285.305,-84.660,175.922,24.646,154.066
C06903=1083.607,285.553,-84.690,175.924,24.649,154.067
C06904=1083.612,285.802,-84.719,175.927,24.653,154.067
C06905=1083.618,286.050,-84.750,175.930,24.657,154.068
C06906=1083.623,286.298,-84.779,175.933,24.660,154.068
C06907=1083.630,286.546,-84.808,175.936,24.664,154.068
C06908=1083.635,286.794,-84.839,175.938,24.667,154.069
C06909=1083.641,287.042,-84.868,175.941,24.671,154.069
C06910=1083.647,287.290,-84.899,175.944,24.675,154.070
C06911=1083.652,287.539,-84.928,175.947,24.678,154.070
C06912=1083.658,287.786,-84.959,175.949,24.681,154.071
C06913=1083.664,288.035,-84.988,175.952,24.685,154.071
C06914=1083.670,288.282,-85.018,175.955,24.689,154.071
C06915=1083.676,288.531,-85.048,175.958,24.692,154.072
C06916=1083.682,288.779,-85.078,175.961,24.696,154.072
C06917=1083.687,289.027,-85.108,175.965,24.699,154.073
C06918=1083.696,289.421,-85.156,175.969,24.705,154.073
C06919=1083.705,289.816,-85.203,175.973,24.711,154.074
C06920=1083.715,290.210,-85.251,175.978,24.717,154.075
C06921=1083.724,290.604,-85.298,175.982,24.722,154.076
C06922=1083.729,290.852,-85.328,175.985,24.726,154.076
C06923=1083.735,291.100,-85.359,175.988,24.729,154.076
C06924=1083.741,291.348,-85.388,175.990,24.733,154.077
C06925=1083.747,291.597,-85.419,175.994,24.737,154.077
C06926=1083.753,291.844,-85.449,175.997,24.740,154.078
C06927=1083.759,292.092,-85.480,175.999,24.744,154.078
C06928=1083.764,292.341,-85.509,176.003,24.748,154.079
C06929=1083.770,292.588,-85.540,176.005,24.751,154.079
C06930=1083.775,292.837,-85.571,176.008,24.755,154.080
C06931=1083.781,293.084,-85.601,176.011,24.758,154.080
C06932=1083.787,293.333,-85.631,176.014,24.762,154.081
C06933=1083.792,293.581,-85.661,176.017,24.766,154.081
C06934=1083.798,293.828,-85.691,176.020,24.770,154.082
C06935=1083.805,294.077,-85.722,176.022,24.773,154.082
C06936=1083.810,294.325,-85.753,176.025,24.777,154.082
C06937=1083.816,294.573,-85.783,176.028,24.781,154.083
C06938=1083.822,294.821,-85.812,176.031,24.784,154.083
C06939=1083.828,295.069,-85.843,176.034,24.788,154.084
C06940=1083.833,295.317,-85.874,176.037,24.792,154.084
C06941=1083.839,295.566,-85.905,176.040,24.796,154.085
C06942=1083.845,295.813,-85.935,176.042,24.799,154.085
C06943=1083.851,296.061,-85.965,176.045,24.802,154.086
C06944=1083.857,296.309,-85.996,176.048,24.806,154.086
C06945=1083.862,296.557,-86.026,176.051,24.810,154.087
C06946=1083.867,296.805,-86.057,176.054,24.814,154.087
C06947=1083.874,297.054,-86.088,176.057,24.817,154.087
C06948=1083.880,297.301,-86.118,176.060,24.821,154.088
C06949=1083.886,297.549,-86.148,176.063,24.825,154.088
C06950=1083.891,297.797,-86.179,176.065,24.828,154.089
C06951=1083.897,298.046,-86.210,176.068,24.832,154.089
C06952=1083.903,298.294,-86.240,176.071,24.836,154.090
C06953=1083.908,298.541,-86.272,176.074,24.840,154.090
C06954=1083.914,298.789,-86.302,176.077,24.843,154.091
C06955=1083.919,299.037,-86.333,176.080,24.847,154.091
C06956=1083.925,299.285,-86.364,176.083,24.851,154.092
C06957=1083.931,299.534,-86.395,176.086,24.855,154.092
C06958=1083.936,299.782,-86.425,176.088,24.858,154.093
C06959=1083.942,300.029,-86.457,176.091,24.862,154.093
C06960=1083.948,300.277,-86.487,176.094,24.866,154.094
C06961=1083.953,300.525,-86.518,176.097,24.870,154.094
C06962=1083.959,300.774,-86.549,176.100,24.874,154.095
C06963=1083.965,301.021,-86.581,176.103,24.878,154.095
C06964=1083.970,301.269,-86.611,176.106,24.881,154.096
C06965=1083.975,301.517,-86.642,176.109,24.885,154.096
C06966=1083.982,301.766,-86.673,176.112,24.889,154.097
C06967=1083.987,302.013,-86.704,176.115,24.893,154.097
C06968=1083.993,302.261,-86.735,176.118,24.897,154.098
C06969=1083.998,302.509,-86.766,176.120,24.901,154.098
C06970=1084.008,302.917,-86.817,176.125,24.907,154.099
C06971=1084.017,303.325,-86.868,176.129,24.913,154.100
C06972=1084.027,303.734,-86.919,176.135,24.919,154.101
C06973=1084.036,304.143,-86.971,176.139,24.926,154.102
C06974=1084.042,304.390,-87.002,176.142,24.930,154.102
C06975=1084.047,304.638,-87.033,176.145,24.934,154.103
C06976=1084.054,304.886,-87.064,176.148,24.938,154.103
C06977=1084.059,305.135,-87.095,176.151,24.941,154.104
C06978=1084.065,305.383,-87.127,176.154,24.945,154.104
C06979=1084.071,305.630,-87.158,176.157,24.949,154.105
C06980=1084.076,305.878,-87.189,176.160,24.953,154.105
C06981=1084.083,306.126,-87.221,176.163,24.957,154.106
C06982=1084.088,306.374,-87.251,176.166,24.961,154.106
C06983=1084.093,306.622,-87.283,176.169,24.965,154.107
C06984=1084.100,306.870,-87.315,176.172,24.969,154.107
C06985=1084.105,307.118,-87.346,176.175,24.972,154.108
C06986=1084.112,307.366,-87.377,176.178,24.976,154.108
C06987=1084.117,307.613,-87.409,176.181,24.980,154.109
C06988=1084.123,307.862,-87.440,176.184,24.984,154.109
C06989=1084.129,308.109,-87.471,176.187,24.988,154.110
C06990=1084.135,308.357,-87.503,176.190,24.992,154.110
C06991=1084.140,308.605,-87.534,176.193,24.995,154.111
C06992=1084.147,308.853,-87.565,176.196,24.999,154.111
C06993=1084.152,309.101,-87.597,176.199,25.003,154.112
C06994=1084.158,309.349,-87.629,176.202,25.007,154.112
C06995=1084.164,309.597,-87.659,176.204,25.011,154.113
C06996=1084.170,309.845,-87.691,176.207,25.015,154.113
C06997=1084.175,310.093,-87.723,176.211,25.019,154.114
C06998=1084.182,310.341,-87.755,176.213,25.022,154.114
C06999=1084.188,310.588,-87.786,176.216,25.026,154.115
C07000=1084.194,310.836,-87.818,176.218,25.030,154.115
C07001=1084.199,311.084,-87.849,176.221,25.034,154.116
C07002=1084.205,311.332,-87.881,176.224,25.038,154.116
C07003=1084.211,311.580,-87.912,176.227,25.042,154.117
C07004=1084.217,311.828,-87.944,176.230,25.046,154.118
C07005=1084.223,312.076,-87.976,176.233,25.050,154.118
C07006=1084.229,312.323,-88.007,176.236,25.054,154.118
C07007=1084.235,312.572,-88.039,176.239,25.058,154.119
C07008=1084.241,312.820,-88.071,176.242,25.062,154.120
C07009=1084.246,313.067,-88.103,176.245,25.066,154.120
C07010=1084.253,313.315,-88.135,176.248,25.069,154.121
C07011=1084.258,313.563,-88.166,176.251,25.073,154.121
C07012=1084.264,313.811,-88.198,176.254,25.077,154.122
C07013=1084.270,314.059,-88.230,176.257,25.081,154.122
C07014=1084.276,314.307,-88.262,176.260,25.085,154.123
C07015=1084.282,314.555,-88.293,176.264,25.090,154.123
C07016=1084.288,314.803,-88.325,176.267,25.093,154.124
C07017=1084.294,315.051,-88.357,176.270,25.098,154.124
C07018=1084.300,315.298,-88.390,176.273,25.102,154.125
C07019=1084.306,315.546,-88.422,176.276,25.106,154.125
C07020=1084.311,315.794,-88.454,176.279,25.109,154.126
C07021=1084.317,316.042,-88.486,176.282,25.114,154.127
C07022=1084.327,316.453,-88.539,176.286,25.121,154.128
C07023=1084.336,316.865,-88.593,176.291,25.127,154.128
C07024=1084.345,317.276,-88.646,176.296,25.134,154.129
C07025=1084.355,317.687,-88.699,176.300,25.141,154.130
C07026=1084.360,317.936,-88.732,176.303,25.145,154.131
C07027=1084.366,318.183,-88.764,176.306,25.149,154.132
C07028=1084.372,318.431,-88.796,176.310,25.154,154.132
C07029=1084.378,318.679,-88.828,176.313,25.158,154.133
C07030=1084.383,318.926,-88.861,176.316,25.162,154.133
C07031=1084.389,319.175,-88.893,176.319,25.166,154.134
C07032=1084.395,319.422,-88.926,176.322,25.170,154.134
C07033=1084.400,319.670,-88.958,176.325,25.174,154.135
C07034=1084.406,319.918,-88.990,176.328,25.178,154.136
C07035=1084.412,320.166,-89.023,176.331,25.183,154.136
C07036=1084.418,320.414,-89.055,176.334,25.187,154.137
C07037=1084.424,320.661,-89.088,176.337,25.191,154.137
C07038=1084.429,320.909,-89.120,176.339,25.195,154.138
C07039=1084.435,321.157,-89.153,176.342,25.199,154.139
C07040=1084.441,321.405,-89.185,176.345,25.204,154.139
C07041=1084.446,321.652,-89.218,176.348,25.207,154.140
C07042=1084.452,321.901,-89.250,176.351,25.211,154.140
C07043=1084.458,322.148,-89.283,176.355,25.216,154.141
C07044=1084.464,322.396,-89.316,176.358,25.220,154.142
C07045=1084.470,322.644,-89.348,176.361,25.225,154.142
C07046=1084.476,322.891,-89.380,176.364,25.229,154.143
C07047=1084.482,323.139,-89.412,176.367,25.233,154.143
C07048=1084.487,323.387,-89.446,176.370,25.237,154.144
C07049=1084.493,323.635,-89.479,176.372,25.241,154.145
C07050=1084.499,323.884,-89.511,176.375,25.245,154.145
C07051=1084.505,324.131,-89.544,176.378,25.250,154.146
C07052=1084.511,324.379,-89.577,176.381,25.254,154.146
C07053=1084.516,324.626,-89.610,176.384,25.258,154.147
C07054=1084.522,324.874,-89.642,176.388,25.262,154.148
C07055=1084.529,325.122,-89.674,176.391,25.267,154.148
C07056=1084.534,325.370,-89.708,176.394,25.271,154.149
C07057=1084.540,325.617,-89.740,176.397,25.275,154.149
C07058=1084.546,325.865,-89.772,176.400,25.279,154.150
C07059=1084.552,326.113,-89.806,176.402,25.284,154.151
C07060=1084.558,326.361,-89.839,176.405,25.288,154.151
C07061=1084.564,326.609,-89.872,176.408,25.292,154.152
C07062=1084.570,326.856,-89.905,176.412,25.297,154.152
C07063=1084.576,327.104,-89.938,176.415,25.301,154.153
C07064=1084.582,327.352,-89.971,176.418,25.305,154.154
C07065=1084.588,327.600,-90.003,176.421,25.309,154.154
C07066=1084.593,327.848,-90.036,176.424,25.314,154.155
C07067=1084.600,328.096,-90.069,176.427,25.318,154.156
C07068=1084.605,328.344,-90.102,176.430,25.322,154.156
C07069=1084.612,328.591,-90.135,176.433,25.327,154.157
C07070=1084.617,328.839,-90.168,176.436,25.331,154.157
C07071=1084.623,329.087,-90.201,176.439,25.335,154.158
C07072=1084.629,329.335,-90.234,176.442,25.339,154.159
C07073=1084.635,329.582,-90.267,176.445,25.344,154.159
C07074=1084.645,329.987,-90.322,176.450,25.351,154.160
C07075=1084.655,330.391,-90.375,176.455,25.358,154.161
C07076=1084.665,330.796,-90.430,176.461,25.365,154.162
C07077=1084.675,331.200,-90.484,176.466,25.372,154.163
C07078=1084.681,331.448,-90.517,176.469,25.377,154.164
C07079=1084.686,331.696,-90.550,176.472,25.381,154.165
C07080=1084.692,331.944,-90.584,176.474,25.385,154.165
C07081=1084.699,332.191,-90.617,176.477,25.390,154.166
C07082=1084.704,332.439,-90.650,176.480,25.394,154.167
C07083=1084.710,332.687,-90.684,176.484,25.399,154.167
C07084=1084.715,332.934,-90.717,176.487,25.403,154.168
C07085=1084.722,333.181,-90.751,176.490,25.408,154.169
C07086=1084.727,333.429,-90.784,176.493,25.412,154.169
C07087=1084.733,333.677,-90.817,176.495,25.416,154.170
C07088=1084.739,333.925,-90.852,176.499,25.421,154.171
C07089=1084.745,334.173,-90.885,176.502,25.426,154.171
C07090=1084.751,334.421,-90.918,176.505,25.430,154.172
C07091=1084.757,334.668,-90.952,176.508,25.435,154.173
C07092=1084.763,334.916,-90.985,176.511,25.440,154.173
C07093=1084.769,335.163,-91.019,176.514,25.444,154.174
C07094=1084.774,335.411,-91.052,176.517,25.448,154.175
C07095=1084.780,335.659,-91.086,176.520,25.453,154.175
C07096=1084.786,335.907,-91.120,176.523,25.457,154.176
C07097=1084.792,336.155,-91.153,176.527,25.462,154.177
C07098=1084.798,336.402,-91.187,176.530,25.466,154.177
C07099=1084.804,336.650,-91.220,176.533,25.471,154.178
C07100=1084.810,336.897,-91.254,176.535,25.476,154.179
C07101=1084.816,337.145,-91.289,176.539,25.480,154.179
C07102=1084.822,337.393,-91.322,176.542,25.485,154.180
C07103=1084.828,337.640,-91.356,176.545,25.489,154.181
C07104=1084.833,337.888,-91.390,176.548,25.494,154.181
C07105=1084.840,338.135,-91.423,176.551,25.499,154.182
C07106=1084.846,338.383,-91.457,176.554,25.503,154.183
C07107=1084.852,338.631,-91.491,176.557,25.508,154.184
C07108=1084.857,338.879,-91.525,176.561,25.513,154.184
C07109=1084.863,339.126,-91.559,176.564,25.517,154.185
C07110=1084.868,339.374,-91.593,176.566,25.522,154.186
C07111=1084.875,339.622,-91.627,176.569,25.527,154.186
C07112=1084.881,339.869,-91.661,176.573,25.531,154.187
C07113=1084.887,340.116,-91.695,176.576,25.536,154.188
C07114=1084.892,340.364,-91.729,176.579,25.541,154.189
C07115=1084.899,340.612,-91.763,176.582,25.546,154.189
C07116=1084.904,340.860,-91.797,176.585,25.550,154.190
C07117=1084.910,341.107,-91.831,176.588,25.555,154.191
C07118=1084.917,341.355,-91.866,176.591,25.560,154.192
C07119=1084.923,341.602,-91.900,176.595,25.565,154.192
C07120=1084.927,341.850,-91.934,176.598,25.569,154.193
C07121=1084.933,342.098,-91.968,176.600,25.574,154.194
C07122=1084.940,342.346,-92.002,176.604,25.579,154.194
C07123=1084.946,342.593,-92.036,176.607,25.584,154.195
C07124=1084.951,342.840,-92.070,176.610,25.588,154.196
C07125=1084.958,343.088,-92.105,176.614,25.593,154.197
C07126=1084.967,343.487,-92.160,176.618,25.601,154.198
C07127=1084.977,343.886,-92.215,176.623,25.608,154.199
C07128=1084.987,344.285,-92.271,176.628,25.616,154.200
C07129=1084.996,344.684,-92.326,176.633,25.624,154.202
C07130=1085.002,344.931,-92.361,176.637,25.629,154.202
C07131=1085.008,345.179,-92.395,176.639,25.634,154.203
C07132=1085.014,345.427,-92.429,176.642,25.639,154.204
C07133=1085.019,345.674,-92.464,176.646,25.644,154.205
C07134=1085.025,345.922,-92.498,176.649,25.649,154.205
C07135=1085.032,346.169,-92.533,176.652,25.653,154.206
C07136=1085.037,346.416,-92.568,176.655,25.658,154.207
C07137=1085.043,346.664,-92.602,176.658,25.663,154.208
C07138=1085.049,346.912,-92.636,176.662,25.668,154.208
C07139=1085.055,347.159,-92.672,176.664,25.673,154.209
C07140=1085.061,347.407,-92.706,176.667,25.678,154.210
C07141=1085.067,347.655,-92.740,176.671,25.683,154.211
C07142=1085.073,347.902,-92.776,176.674,25.688,154.212
C07143=1085.079,348.149,-92.810,176.677,25.693,154.212
C07144=1085.084,348.397,-92.845,176.680,25.698,154.213
C07145=1085.091,348.644,-92.879,176.683,25.703,154.214
C07146=1085.096,348.892,-92.915,176.687,25.708,154.215
C07147=1085.102,349.139,-92.949,176.690,25.713,154.216
C07148=1085.109,349.387,-92.984,176.692,25.718,154.216
C07149=1085.114,349.634,-93.018,176.696,25.723,154.217
C07150=1085.121,349.882,-93.053,176.699,25.728,154.218
C07151=1085.126,350.129,-93.088,176.703,25.733,154.219
C07152=1085.133,350.377,-93.123,176.705,25.738,154.220
C07153=1085.138,350.624,-93.158,176.708,25.744,154.221
C07154=1085.145,350.872,-93.193,176.712,25.749,154.221
C07155=1085.150,351.119,-93.228,176.714,25.754,154.222
C07156=1085.157,351.367,-93.263,176.718,25.759,154.223
C07157=1085.162,351.614,-93.297,176.721,25.764,154.224
C07158=1085.168,351.862,-93.333,176.725,25.769,154.224
C07159=1085.174,352.109,-93.368,176.727,25.774,154.225
C07160=1085.180,352.357,-93.403,176.730,25.779,154.226
C07161=1085.186,352.604,-93.438,176.734,25.784,154.227
C07162=1085.192,352.851,-93.473,176.737,25.789,154.228
C07163=1085.198,353.099,-93.508,176.740,25.795,154.229
C07164=1085.204,353.347,-93.544,176.743,25.800,154.229
C07165=1085.210,353.594,-93.579,176.747,25.805,154.230
C07166=1085.216,353.842,-93.613,176.749,25.810,154.231
C07167=1085.222,354.089,-93.649,176.753,25.816,154.232
C07168=1085.228,354.336,-93.685,176.756,25.821,154.233
C07169=1085.234,354.583,-93.719,176.759,25.826,154.234
C07170=1085.240,354.831,-93.755,176.762,25.831,154.235
C07171=1085.246,355.079,-93.790,176.765,25.837,154.236
C07172=1085.251,355.326,-93.825,176.769,25.842,154.236
C07173=1085.258,355.573,-93.861,176.771,25.847,154.237
C07174=1085.264,355.821,-93.896,176.775,25.852,154.238
C07175=1085.269,356.068,-93.932,176.778,25.858,154.239
C07176=1085.275,356.316,-93.967,176.781,25.863,154.240
C07177=1085.282,356.563,-94.002,176.784,25.868,154.241
C07178=1085.291,356.964,-94.060,176.789,25.877,154.242
C07179=1085.301,357.366,-94.117,176.795,25.886,154.244
C07180=1085.311,357.768,-94.175,176.800,25.894,154.245
C07181=1085.320,358.170,-94.233,176.805,25.903,154.246
C07182=1085.327,358.417,-94.269,176.808,25.908,154.247
C07183=1085.333,358.665,-94.305,176.811,25.914,154.248
C07184=1085.339,358.913,-94.340,176.815,25.919,154.249
C07185=1085.344,359.159,-94.376,176.817,25.925,154.250
C07186=1085.351,359.407,-94.411,176.821,25.930,154.251
C07187=1085.357,359.655,-94.447,176.825,25.935,154.252
C07188=1085.363,359.902,-94.482,176.827,25.941,154.253
C07189=1085.369,360.149,-94.519,176.831,25.946,154.254
C07190=1085.375,360.396,-94.554,176.834,25.952,154.255
C07191=1085.381,360.644,-94.590,176.837,25.957,154.256
C07192=1085.387,360.892,-94.626,176.840,25.963,154.256
C07193=1085.393,361.139,-94.662,176.844,25.968,154.257
C07194=1085.398,361.386,-94.697,176.846,25.974,154.258
C07195=1085.404,361.633,-94.733,176.850,25.979,154.259
C07196=1085.411,361.880,-94.770,176.853,25.985,154.260
C07197=1085.417,362.128,-94.805,176.856,25.991,154.261
C07198=1085.423,362.375,-94.842,176.859,25.996,154.262
C07199=1085.429,362.622,-94.877,176.863,26.002,154.263
C07200=1085.435,362.870,-94.913,176.866,26.007,154.264
C07201=1085.441,363.117,-94.949,176.869,26.013,154.265
C07202=1085.447,363.364,-94.985,176.872,26.019,154.266
C07203=1085.453,363.611,-95.022,176.875,26.024,154.267
C07204=1085.459,363.859,-95.057,176.879,26.030,154.268
C07205=1085.466,364.106,-95.094,176.881,26.036,154.269
C07206=1085.471,364.353,-95.129,176.885,26.041,154.270
C07207=1085.477,364.600,-95.166,176.889,26.047,154.271
C07208=1085.483,364.848,-95.202,176.891,26.053,154.272
C07209=1085.489,365.095,-95.238,176.895,26.058,154.273
C07210=1085.495,365.342,-95.275,176.898,26.064,154.274
C07211=1085.501,365.590,-95.310,176.901,26.070,154.275
C07212=1085.508,365.837,-95.347,176.905,26.076,154.276
C07213=1085.513,366.084,-95.384,176.907,26.081,154.277
C07214=1085.519,366.331,-95.419,176.911,26.087,154.278
C07215=1085.525,366.578,-95.456,176.914,26.093,154.279
C07216=1085.532,366.826,-95.492,176.917,26.099,154.280
C07217=1085.537,367.073,-95.529,176.921,26.105,154.281
C07218=1085.543,367.321,-95.565,176.923,26.110,154.282
C07219=1085.549,367.568,-95.601,176.927,26.116,154.283
C07220=1085.555,367.815,-95.638,176.931,26.122,154.284
C07221=1085.561,368.062,-95.675,176.933,26.128,154.285
C07222=1085.568,368.309,-95.711,176.937,26.134,154.286
C07223=1085.573,368.556,-95.748,176.939,26.140,154.287
C07224=1085.579,368.804,-95.784,176.943,26.145,154.288
C07225=1085.586,369.051,-95.821,176.947,26.152,154.289
C07226=1085.591,369.299,-95.858,176.949,26.157,154.290
C07227=1085.598,369.546,-95.894,176.953,26.163,154.291
C07228=1085.604,369.793,-95.930,176.956,26.170,154.292
C07229=1085.610,370.040,-95.968,176.959,26.175,154.293
C07230=1085.620,370.457,-96.030,176.964,26.185,154.295
C07231=1085.630,370.875,-96.091,176.970,26.195,154.297
C07232=1085.641,371.292,-96.154,176.976,26.206,154.298
C07233=1085.651,371.710,-96.215,176.981,26.216,154.300
C07234=1085.657,371.957,-96.253,176.985,26.222,154.301
C07235=1085.663,372.204,-96.289,176.987,26.228,154.302
C07236=1085.669,372.452,-96.327,176.991,26.234,154.303
C07237=1085.676,372.699,-96.363,176.994,26.240,154.305
C07238=1085.682,372.946,-96.400,176.997,26.246,154.306
C07239=1085.688,373.193,-96.437,177.001,26.252,154.307
C07240=1085.694,373.440,-96.474,177.004,26.258,154.308
C07241=1085.700,373.687,-96.511,177.008,26.265,154.309
C07242=1085.706,373.934,-96.547,177.010,26.271,154.310
C07243=1085.712,374.181,-96.585,177.014,26.277,154.311
C07244=1085.719,374.429,-96.622,177.017,26.283,154.312
C07245=1085.725,374.676,-96.659,177.020,26.290,154.313
C07246=1085.730,374.923,-96.697,177.023,26.296,154.314
C07247=1085.736,375.170,-96.734,177.027,26.302,154.316
C07248=1085.743,375.416,-96.771,177.030,26.309,154.317
C07249=1085.748,375.664,-96.808,177.033,26.314,154.318
C07250=1085.754,375.911,-96.846,177.036,26.321,154.319
C07251=1085.761,376.158,-96.882,177.040,26.328,154.320
C07252=1085.767,376.405,-96.920,177.043,26.334,154.321
C07253=1085.773,376.652,-96.957,177.046,26.340,154.322
C07254=1085.779,376.899,-96.994,177.049,26.346,154.324
C07255=1085.785,377.146,-97.031,177.053,26.353,154.325
C07256=1085.791,377.393,-97.069,177.056,26.360,154.326
C07257=1085.797,377.641,-97.107,177.060,26.366,154.327
C07258=1085.804,377.887,-97.144,177.063,26.372,154.328
C07259=1085.810,378.134,-97.182,177.066,26.378,154.329
C07260=1085.815,378.382,-97.219,177.070,26.385,154.330
C07261=1085.822,378.629,-97.257,177.073,26.391,154.332
C07262=1085.828,378.875,-97.294,177.076,26.398,154.333
C07263=1085.834,379.122,-97.332,177.079,26.404,154.334
C07264=1085.840,379.370,-97.369,177.083,26.411,154.335
C07265=1085.846,379.617,-97.407,177.086,26.417,154.336
C07266=1085.853,379.863,-97.444,177.089,26.424,154.338
C07267=1085.859,380.110,-97.482,177.092,26.430,154.339
C07268=1085.864,380.358,-97.519,177.095,26.437,154.340
C07269=1085.871,380.605,-97.557,177.099,26.444,154.341
C07270=1085.877,380.852,-97.595,177.102,26.450,154.342
C07271=1085.884,381.098,-97.632,177.106,26.457,154.344
C07272=1085.890,381.346,-97.670,177.109,26.464,154.345
C07273=1085.896,381.592,-97.708,177.112,26.470,154.346
C07274=1085.902,381.840,-97.746,177.115,26.476,154.347
C07275=1085.908,382.087,-97.784,177.119,26.483,154.349
C07276=1085.914,382.333,-97.821,177.122,26.490,154.350
